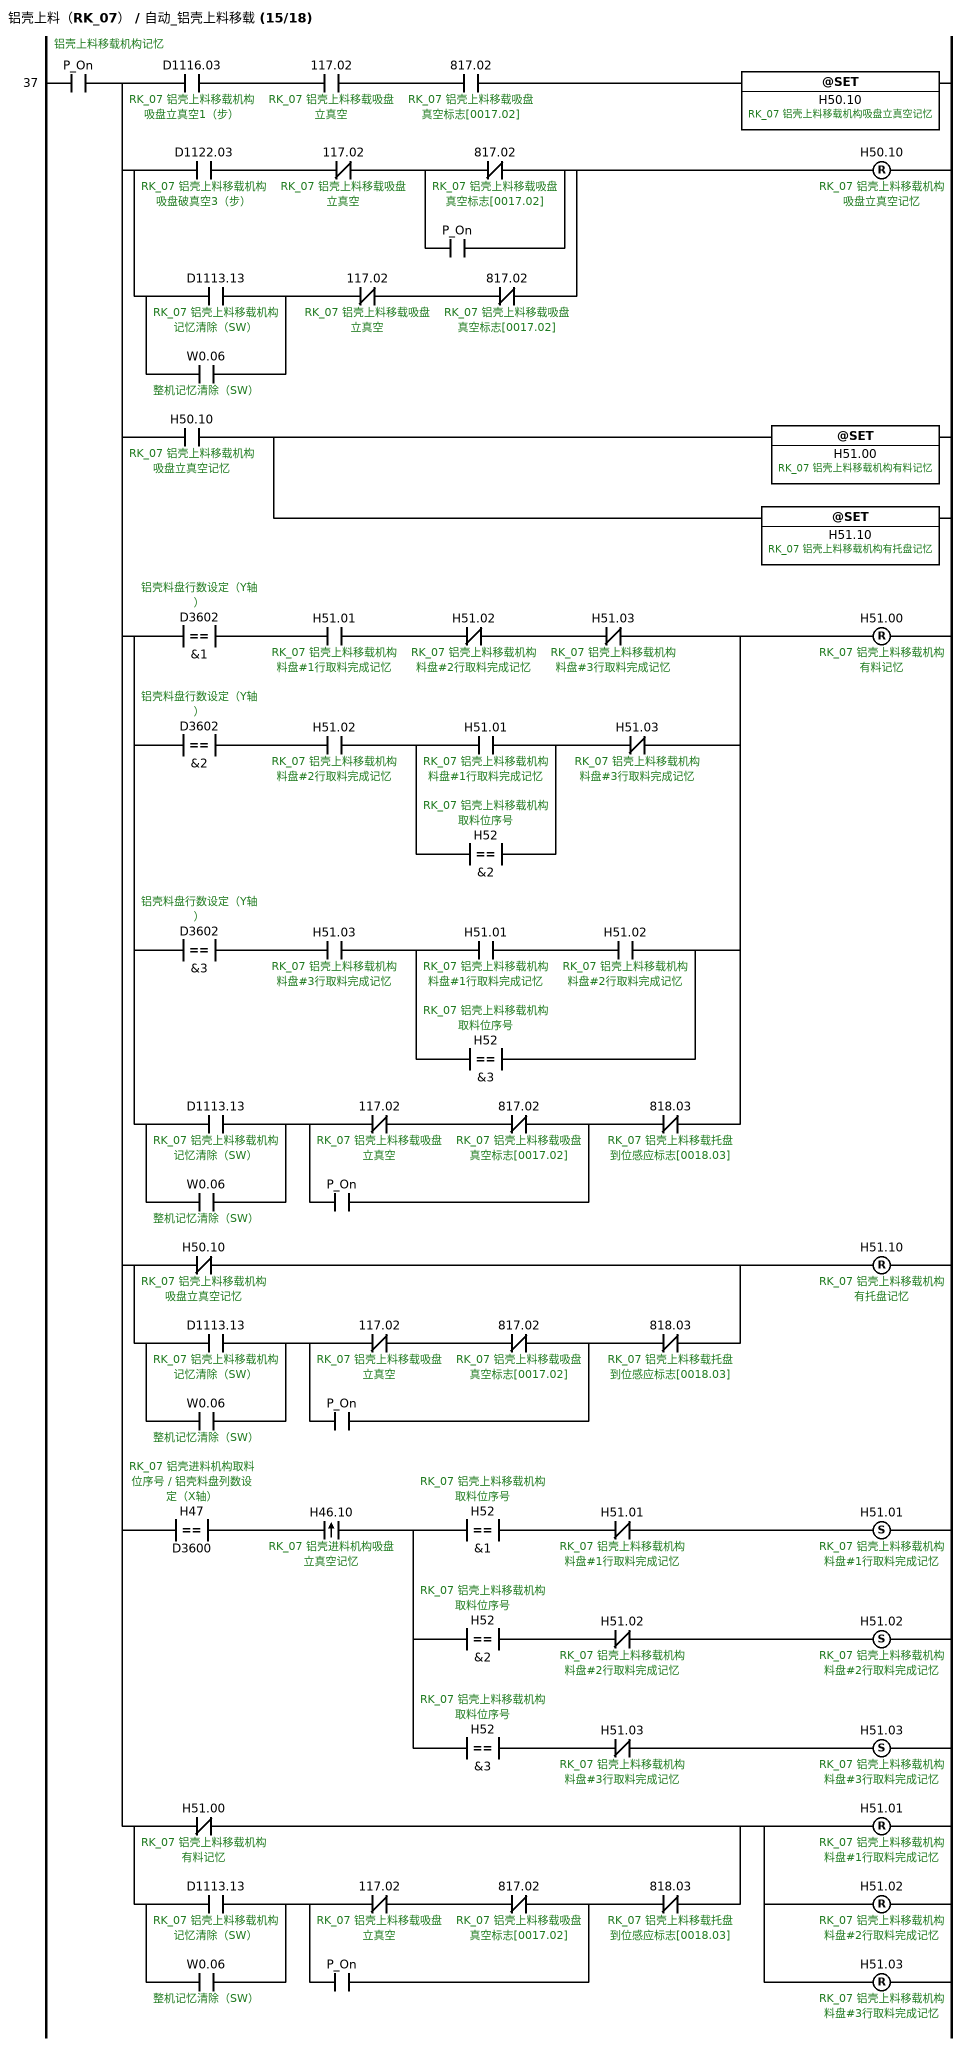
; [picture p600: 铝壳上料（RK_07） / 自动_铝壳上料移载, rungs 37-37]
; rung 37: 铝壳上料移载机构记忆
LD P_On
OUT TR0
AND D1116.03  ; RK_07 铝壳上料移载机构吸盘立真空1（步）
AND 117.02  ; RK_07 铝壳上料移载吸盘立真空
AND 817.02  ; RK_07 铝壳上料移载吸盘真空标志[0017.02]
@SET H50.10  ; RK_07 铝壳上料移载机构吸盘立真空记忆
LD TR0
LD D1122.03  ; RK_07 铝壳上料移载机构吸盘破真空3（步）
ANDNOT 117.02  ; RK_07 铝壳上料移载吸盘立真空
LDNOT 817.02  ; RK_07 铝壳上料移载吸盘真空标志[0017.02]
OR P_On
ANDLD
LD D1113.13  ; RK_07 铝壳上料移载机构记忆清除（SW）
OR W0.06  ; 整机记忆清除（SW）
ANDNOT 117.02  ; RK_07 铝壳上料移载吸盘立真空
ANDNOT 817.02  ; RK_07 铝壳上料移载吸盘真空标志[0017.02]
ORLD
ANDLD
RSET H50.10  ; RK_07 铝壳上料移载机构吸盘立真空记忆
LD TR0
AND H50.10  ; RK_07 铝壳上料移载机构吸盘立真空记忆
@SET H51.00  ; RK_07 铝壳上料移载机构有料记忆
@SET H51.10  ; RK_07 铝壳上料移载机构有托盘记忆
LD TR0
LD=(300) D3602 &1  ; 铝壳料盘行数设定（Y轴）
AND H51.01  ; RK_07 铝壳上料移载机构料盘#1行取料完成记忆
ANDNOT H51.02  ; RK_07 铝壳上料移载机构料盘#2行取料完成记忆
ANDNOT H51.03  ; RK_07 铝壳上料移载机构料盘#3行取料完成记忆
LD=(300) D3602 &2  ; 铝壳料盘行数设定（Y轴）
AND H51.02  ; RK_07 铝壳上料移载机构料盘#2行取料完成记忆
LD H51.01  ; RK_07 铝壳上料移载机构料盘#1行取料完成记忆
OR=(300) H52 &2  ; RK_07 铝壳上料移载机构取料位序号
ANDLD
ANDNOT H51.03  ; RK_07 铝壳上料移载机构料盘#3行取料完成记忆
ORLD
LD=(300) D3602 &3  ; 铝壳料盘行数设定（Y轴）
AND H51.03  ; RK_07 铝壳上料移载机构料盘#3行取料完成记忆
LD H51.01  ; RK_07 铝壳上料移载机构料盘#1行取料完成记忆
AND H51.02  ; RK_07 铝壳上料移载机构料盘#2行取料完成记忆
OR=(300) H52 &3  ; RK_07 铝壳上料移载机构取料位序号
ANDLD
ORLD
LD D1113.13  ; RK_07 铝壳上料移载机构记忆清除（SW）
OR W0.06  ; 整机记忆清除（SW）
LDNOT 117.02  ; RK_07 铝壳上料移载吸盘立真空
ANDNOT 817.02  ; RK_07 铝壳上料移载吸盘真空标志[0017.02]
OR P_On
ANDLD
ANDNOT 818.03  ; RK_07 铝壳上料移载托盘到位感应标志[0018.03]
ORLD
ANDLD
RSET H51.00  ; RK_07 铝壳上料移载机构有料记忆
LD TR0
LDNOT H50.10  ; RK_07 铝壳上料移载机构吸盘立真空记忆
LD D1113.13  ; RK_07 铝壳上料移载机构记忆清除（SW）
OR W0.06  ; 整机记忆清除（SW）
LDNOT 117.02  ; RK_07 铝壳上料移载吸盘立真空
ANDNOT 817.02  ; RK_07 铝壳上料移载吸盘真空标志[0017.02]
OR P_On
ANDLD
ANDNOT 818.03  ; RK_07 铝壳上料移载托盘到位感应标志[0018.03]
ORLD
ANDLD
RSET H51.10  ; RK_07 铝壳上料移载机构有托盘记忆
LD TR0
AND=(300) H47 D3600  ; RK_07 铝壳进料机构取料位序号, 铝壳料盘列数设定（X轴）
@AND H46.10  ; RK_07 铝壳进料机构吸盘立真空记忆
OUT TR1
AND=(300) H52 &1  ; RK_07 铝壳上料移载机构取料位序号
ANDNOT H51.01  ; RK_07 铝壳上料移载机构料盘#1行取料完成记忆
SET H51.01  ; RK_07 铝壳上料移载机构料盘#1行取料完成记忆
LD TR1
AND=(300) H52 &2  ; RK_07 铝壳上料移载机构取料位序号
ANDNOT H51.02  ; RK_07 铝壳上料移载机构料盘#2行取料完成记忆
SET H51.02  ; RK_07 铝壳上料移载机构料盘#2行取料完成记忆
LD TR1
AND=(300) H52 &3  ; RK_07 铝壳上料移载机构取料位序号
ANDNOT H51.03  ; RK_07 铝壳上料移载机构料盘#3行取料完成记忆
SET H51.03  ; RK_07 铝壳上料移载机构料盘#3行取料完成记忆
LD TR0
LDNOT H51.00  ; RK_07 铝壳上料移载机构有料记忆
LD D1113.13  ; RK_07 铝壳上料移载机构记忆清除（SW）
OR W0.06  ; 整机记忆清除（SW）
LDNOT 117.02  ; RK_07 铝壳上料移载吸盘立真空
ANDNOT 817.02  ; RK_07 铝壳上料移载吸盘真空标志[0017.02]
OR P_On
ANDLD
ANDNOT 818.03  ; RK_07 铝壳上料移载托盘到位感应标志[0018.03]
ORLD
ANDLD
RSET H51.01  ; RK_07 铝壳上料移载机构料盘#1行取料完成记忆
RSET H51.02  ; RK_07 铝壳上料移载机构料盘#2行取料完成记忆
RSET H51.03  ; RK_07 铝壳上料移载机构料盘#3行取料完成记忆

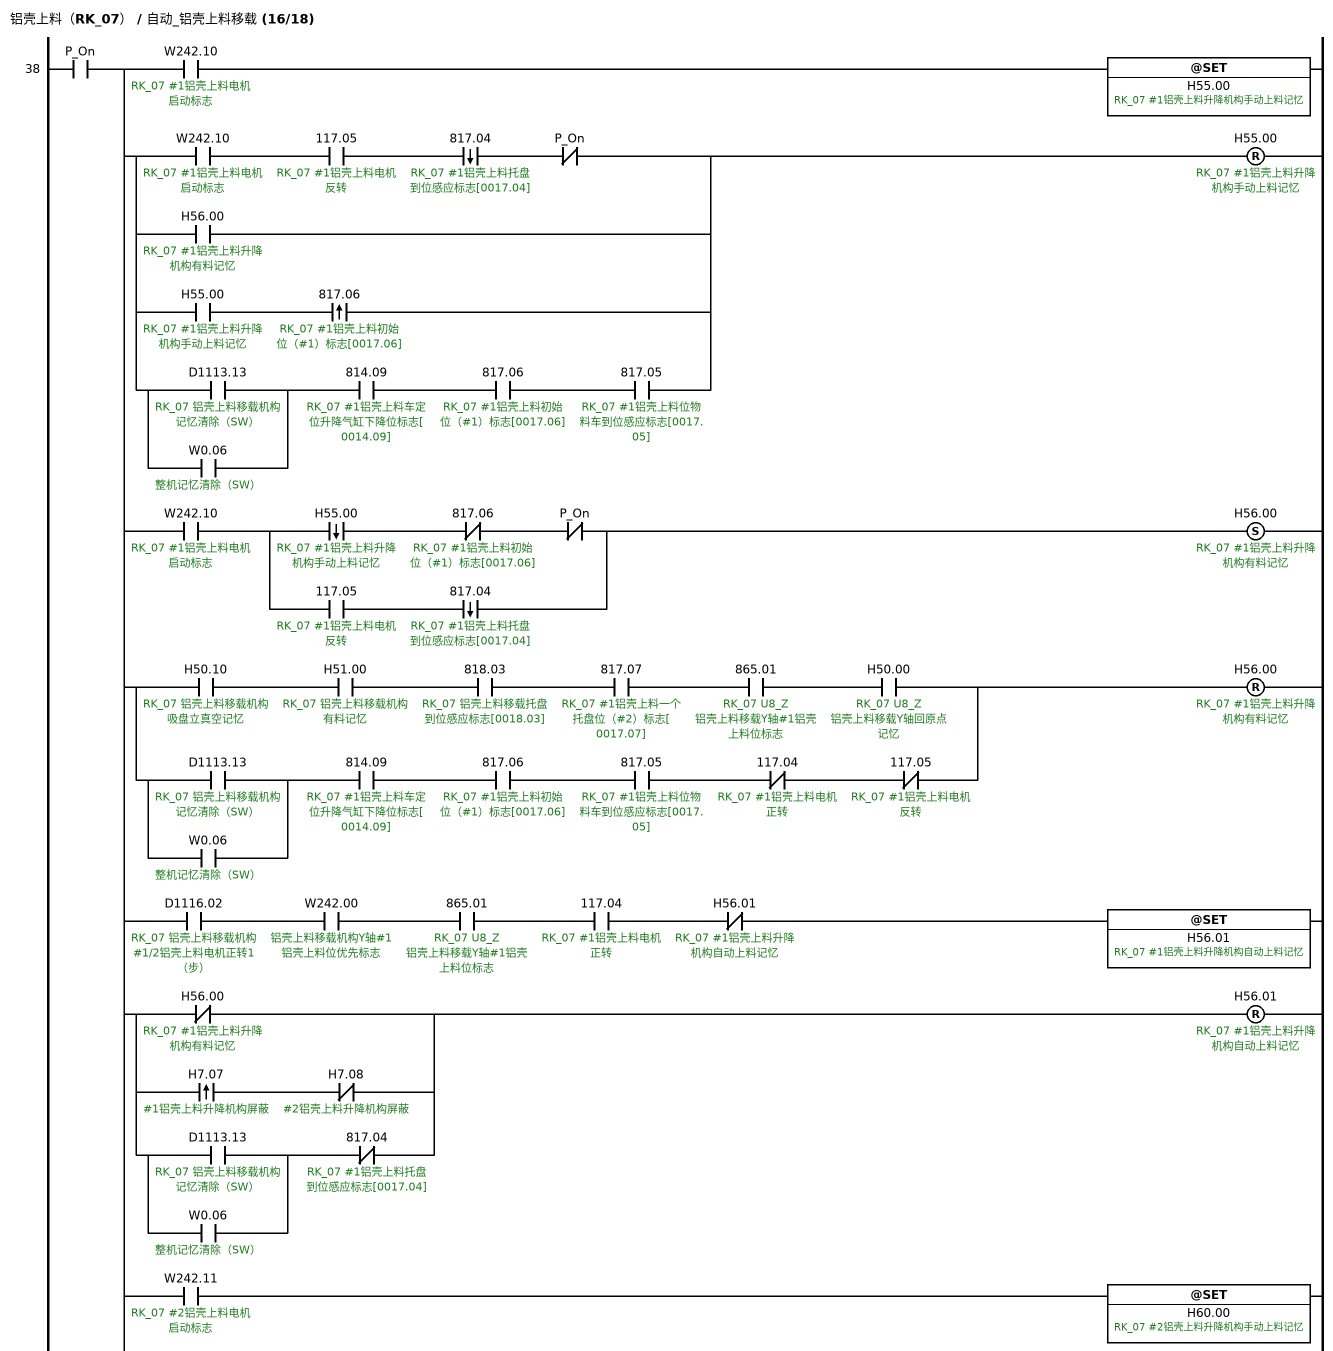

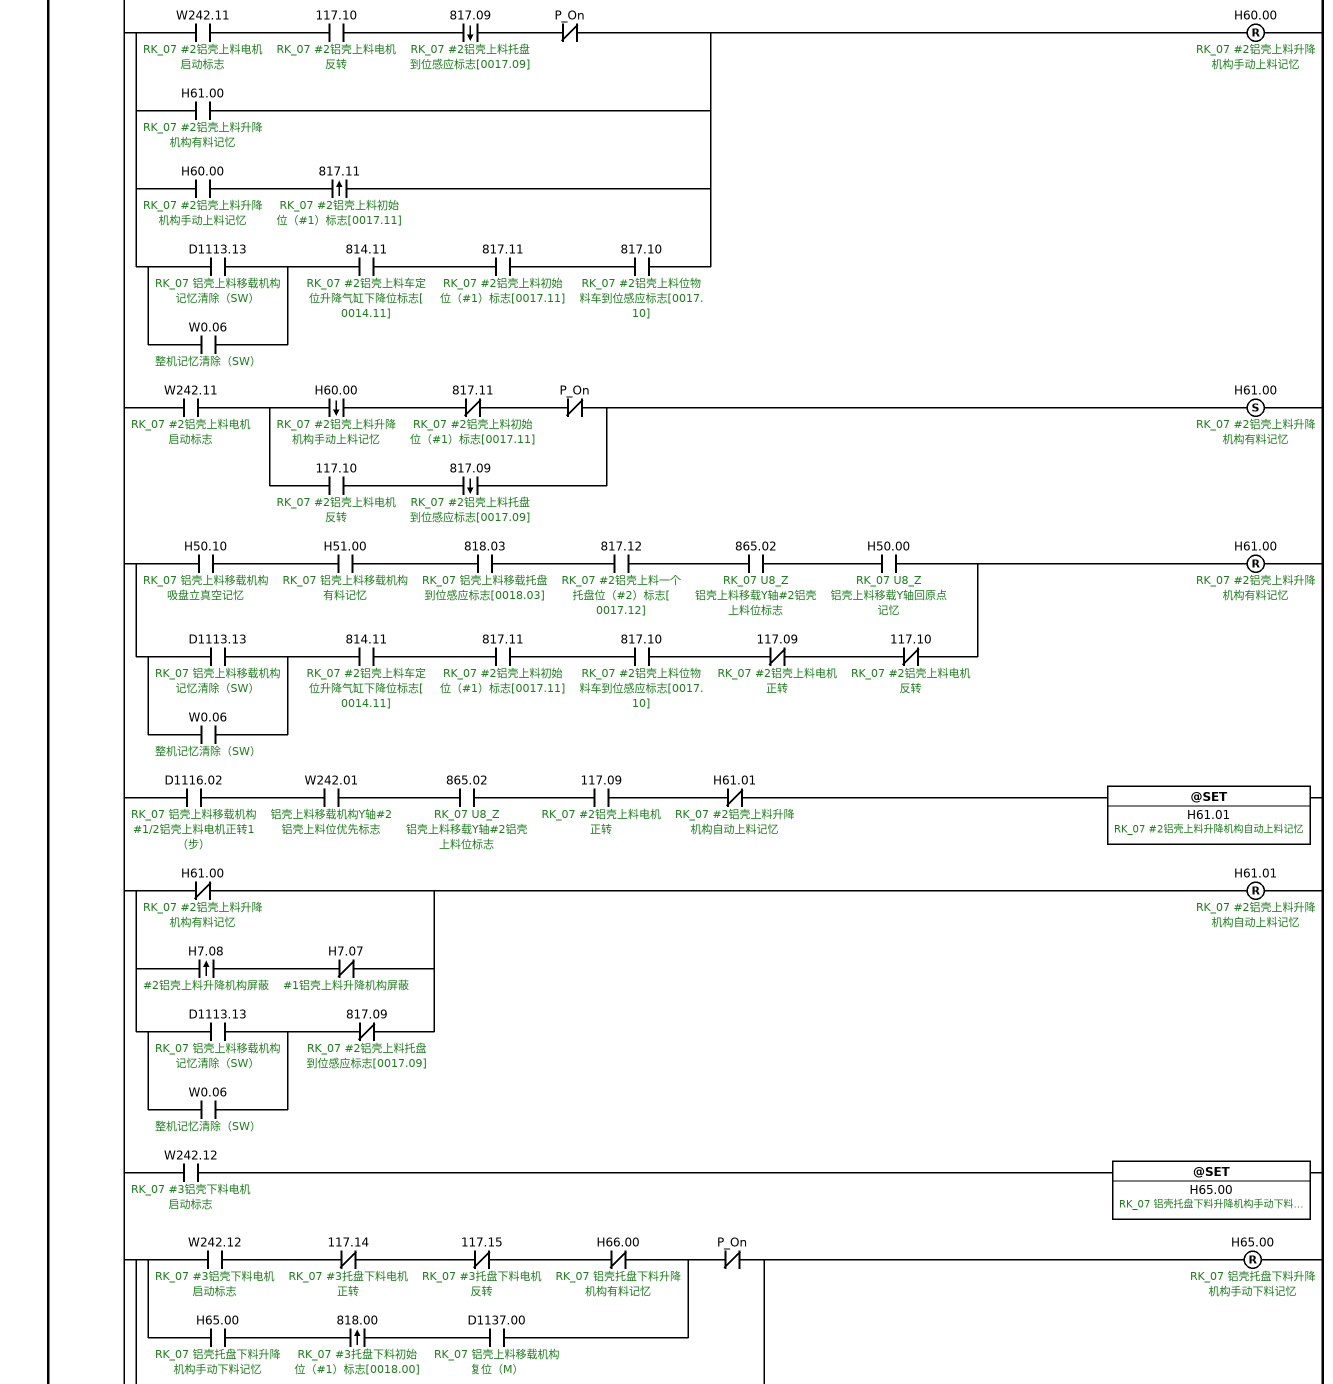

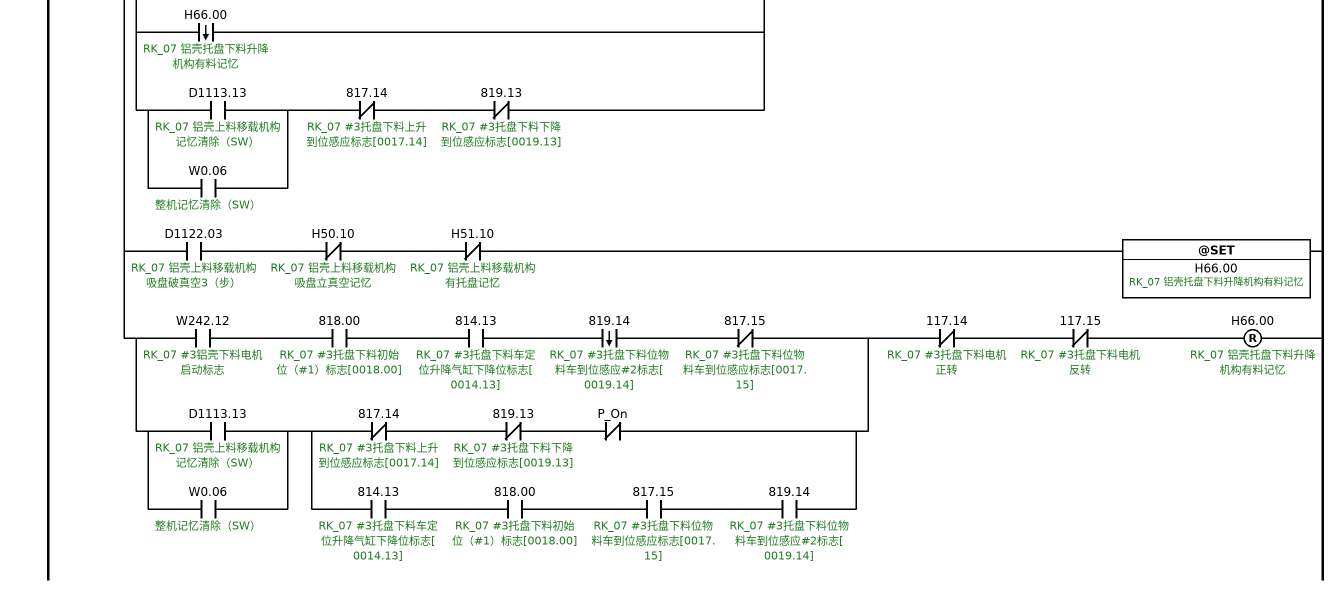
; rung 38
LD P_On
OUT TR0
AND W242.10  ; RK_07 #1铝壳上料电机启动标志
@SET H55.00  ; RK_07 #1铝壳上料升降机构手动上料记忆
LD TR0
LD W242.10  ; RK_07 #1铝壳上料电机启动标志
AND 117.05  ; RK_07 #1铝壳上料电机反转
%AND 817.04  ; RK_07 #1铝壳上料托盘到位感应标志[0017.04]
ANDNOT P_On
OR H56.00  ; RK_07 #1铝壳上料升降机构有料记忆
LD H55.00  ; RK_07 #1铝壳上料升降机构手动上料记忆
@AND 817.06  ; RK_07 #1铝壳上料初始位（#1）标志[0017.06]
ORLD
LD D1113.13  ; RK_07 铝壳上料移载机构记忆清除（SW）
OR W0.06  ; 整机记忆清除（SW）
AND 814.09  ; RK_07 #1铝壳上料车定位升降气缸下降位标志[0014.09]
AND 817.06  ; RK_07 #1铝壳上料初始位（#1）标志[0017.06]
AND 817.05  ; RK_07 #1铝壳上料位物料车到位感应标志[0017.05]
ORLD
ANDLD
RSET H55.00  ; RK_07 #1铝壳上料升降机构手动上料记忆
LD TR0
AND W242.10  ; RK_07 #1铝壳上料电机启动标志
%LD H55.00  ; RK_07 #1铝壳上料升降机构手动上料记忆
ANDNOT 817.06  ; RK_07 #1铝壳上料初始位（#1）标志[0017.06]
ANDNOT P_On
LD 117.05  ; RK_07 #1铝壳上料电机反转
%AND 817.04  ; RK_07 #1铝壳上料托盘到位感应标志[0017.04]
ORLD
ANDLD
SET H56.00  ; RK_07 #1铝壳上料升降机构有料记忆
LD TR0
LD H50.10  ; RK_07 铝壳上料移载机构吸盘立真空记忆
AND H51.00  ; RK_07 铝壳上料移载机构有料记忆
AND 818.03  ; RK_07 铝壳上料移载托盘到位感应标志[0018.03]
AND 817.07  ; RK_07 #1铝壳上料一个托盘位（#2）标志[0017.07]
AND 865.01  ; RK_07 U8_Z 铝壳上料移载Y轴#1铝壳上料位标志
AND H50.00  ; RK_07 U8_Z 铝壳上料移载Y轴回原点记忆
LD D1113.13  ; RK_07 铝壳上料移载机构记忆清除（SW）
OR W0.06  ; 整机记忆清除（SW）
AND 814.09  ; RK_07 #1铝壳上料车定位升降气缸下降位标志[0014.09]
AND 817.06  ; RK_07 #1铝壳上料初始位（#1）标志[0017.06]
AND 817.05  ; RK_07 #1铝壳上料位物料车到位感应标志[0017.05]
ANDNOT 117.04  ; RK_07 #1铝壳上料电机正转
ANDNOT 117.05  ; RK_07 #1铝壳上料电机反转
ORLD
ANDLD
RSET H56.00  ; RK_07 #1铝壳上料升降机构有料记忆
LD TR0
AND D1116.02  ; RK_07 铝壳上料移载机构#1/2铝壳上料电机正转1（步）
AND W242.00  ; 铝壳上料移载机构Y轴#1铝壳上料位优先标志
AND 865.01  ; RK_07 U8_Z 铝壳上料移载Y轴#1铝壳上料位标志
AND 117.04  ; RK_07 #1铝壳上料电机正转
ANDNOT H56.01  ; RK_07 #1铝壳上料升降机构自动上料记忆
@SET H56.01  ; RK_07 #1铝壳上料升降机构自动上料记忆
LD TR0
LDNOT H56.00  ; RK_07 #1铝壳上料升降机构有料记忆
@LD H7.07  ; #1铝壳上料升降机构屏蔽
ANDNOT H7.08  ; #2铝壳上料升降机构屏蔽
ORLD
LD D1113.13  ; RK_07 铝壳上料移载机构记忆清除（SW）
OR W0.06  ; 整机记忆清除（SW）
ANDNOT 817.04  ; RK_07 #1铝壳上料托盘到位感应标志[0017.04]
ORLD
ANDLD
RSET H56.01  ; RK_07 #1铝壳上料升降机构自动上料记忆
LD TR0
AND W242.11  ; RK_07 #2铝壳上料电机启动标志
@SET H60.00  ; RK_07 #2铝壳上料升降机构手动上料记忆
LD TR0
LD W242.11  ; RK_07 #2铝壳上料电机启动标志
AND 117.10  ; RK_07 #2铝壳上料电机反转
%AND 817.09  ; RK_07 #2铝壳上料托盘到位感应标志[0017.09]
ANDNOT P_On
OR H61.00  ; RK_07 #2铝壳上料升降机构有料记忆
LD H60.00  ; RK_07 #2铝壳上料升降机构手动上料记忆
@AND 817.11  ; RK_07 #2铝壳上料初始位（#1）标志[0017.11]
ORLD
LD D1113.13  ; RK_07 铝壳上料移载机构记忆清除（SW）
OR W0.06  ; 整机记忆清除（SW）
AND 814.11  ; RK_07 #2铝壳上料车定位升降气缸下降位标志[0014.11]
AND 817.11  ; RK_07 #2铝壳上料初始位（#1）标志[0017.11]
AND 817.10  ; RK_07 #2铝壳上料位物料车到位感应标志[0017.10]
ORLD
ANDLD
RSET H60.00  ; RK_07 #2铝壳上料升降机构手动上料记忆
LD TR0
AND W242.11  ; RK_07 #2铝壳上料电机启动标志
%LD H60.00  ; RK_07 #2铝壳上料升降机构手动上料记忆
ANDNOT 817.11  ; RK_07 #2铝壳上料初始位（#1）标志[0017.11]
ANDNOT P_On
LD 117.10  ; RK_07 #2铝壳上料电机反转
%AND 817.09  ; RK_07 #2铝壳上料托盘到位感应标志[0017.09]
ORLD
ANDLD
SET H61.00  ; RK_07 #2铝壳上料升降机构有料记忆
LD TR0
LD H50.10  ; RK_07 铝壳上料移载机构吸盘立真空记忆
AND H51.00  ; RK_07 铝壳上料移载机构有料记忆
AND 818.03  ; RK_07 铝壳上料移载托盘到位感应标志[0018.03]
AND 817.12  ; RK_07 #2铝壳上料一个托盘位（#2）标志[0017.12]
AND 865.02  ; RK_07 U8_Z 铝壳上料移载Y轴#2铝壳上料位标志
AND H50.00  ; RK_07 U8_Z 铝壳上料移载Y轴回原点记忆
LD D1113.13  ; RK_07 铝壳上料移载机构记忆清除（SW）
OR W0.06  ; 整机记忆清除（SW）
AND 814.11  ; RK_07 #2铝壳上料车定位升降气缸下降位标志[0014.11]
AND 817.11  ; RK_07 #2铝壳上料初始位（#1）标志[0017.11]
AND 817.10  ; RK_07 #2铝壳上料位物料车到位感应标志[0017.10]
ANDNOT 117.09  ; RK_07 #2铝壳上料电机正转
ANDNOT 117.10  ; RK_07 #2铝壳上料电机反转
ORLD
ANDLD
RSET H61.00  ; RK_07 #2铝壳上料升降机构有料记忆
LD TR0
AND D1116.02  ; RK_07 铝壳上料移载机构#1/2铝壳上料电机正转1（步）
AND W242.01  ; 铝壳上料移载机构Y轴#2铝壳上料位优先标志
AND 865.02  ; RK_07 U8_Z 铝壳上料移载Y轴#2铝壳上料位标志
AND 117.09  ; RK_07 #2铝壳上料电机正转
ANDNOT H61.01  ; RK_07 #2铝壳上料升降机构自动上料记忆
@SET H61.01  ; RK_07 #2铝壳上料升降机构自动上料记忆
LD TR0
LDNOT H61.00  ; RK_07 #2铝壳上料升降机构有料记忆
@LD H7.08  ; #2铝壳上料升降机构屏蔽
ANDNOT H7.07  ; #1铝壳上料升降机构屏蔽
ORLD
LD D1113.13  ; RK_07 铝壳上料移载机构记忆清除（SW）
OR W0.06  ; 整机记忆清除（SW）
ANDNOT 817.09  ; RK_07 #2铝壳上料托盘到位感应标志[0017.09]
ORLD
ANDLD
RSET H61.01  ; RK_07 #2铝壳上料升降机构自动上料记忆
LD TR0
AND W242.12  ; RK_07 #3铝壳下料电机启动标志
@SET H65.00  ; RK_07 铝壳托盘下料升降机构手动下料记忆
LD TR0
LD W242.12  ; RK_07 #3铝壳下料电机启动标志
ANDNOT 117.14  ; RK_07 #3托盘下料电机正转
ANDNOT 117.15  ; RK_07 #3托盘下料电机反转
ANDNOT H66.00  ; RK_07 铝壳托盘下料升降机构有料记忆
LD H65.00  ; RK_07 铝壳托盘下料升降机构手动下料记忆
@AND 818.00  ; RK_07 #3托盘下料初始位（#1）标志[0018.00]
AND D1137.00  ; RK_07 铝壳上料移载机构复位（M）
ORLD
ANDNOT P_On
%OR H66.00  ; RK_07 铝壳托盘下料升降机构有料记忆
LD D1113.13  ; RK_07 铝壳上料移载机构记忆清除（SW）
OR W0.06  ; 整机记忆清除（SW）
ANDNOT 817.14  ; RK_07 #3托盘下料上升到位感应标志[0017.14]
ANDNOT 819.13  ; RK_07 #3托盘下料下降到位感应标志[0019.13]
ORLD
ANDLD
RSET H65.00  ; RK_07 铝壳托盘下料升降机构手动下料记忆
LD TR0
AND D1122.03  ; RK_07 铝壳上料移载机构吸盘破真空3（步）
ANDNOT H50.10  ; RK_07 铝壳上料移载机构吸盘立真空记忆
ANDNOT H51.10  ; RK_07 铝壳上料移载机构有托盘记忆
@SET H66.00  ; RK_07 铝壳托盘下料升降机构有料记忆
LD TR0
LD W242.12  ; RK_07 #3铝壳下料电机启动标志
AND 818.00  ; RK_07 #3托盘下料初始位（#1）标志[0018.00]
AND 814.13  ; RK_07 #3托盘下料车定位升降气缸下降位标志[0014.13]
%AND 819.14  ; RK_07 #3托盘下料位物料车到位感应#2标志[0019.14]
ANDNOT 817.15  ; RK_07 #3托盘下料位物料车到位感应标志[0017.15]
LD D1113.13  ; RK_07 铝壳上料移载机构记忆清除（SW）
OR W0.06  ; 整机记忆清除（SW）
LDNOT 817.14  ; RK_07 #3托盘下料上升到位感应标志[0017.14]
ANDNOT 819.13  ; RK_07 #3托盘下料下降到位感应标志[0019.13]
ANDNOT P_On
LD 814.13  ; RK_07 #3托盘下料车定位升降气缸下降位标志[0014.13]
AND 818.00  ; RK_07 #3托盘下料初始位（#1）标志[0018.00]
AND 817.15  ; RK_07 #3托盘下料位物料车到位感应标志[0017.15]
AND 819.14  ; RK_07 #3托盘下料位物料车到位感应#2标志[0019.14]
ORLD
ANDLD
ORLD
ANDLD
ANDNOT 117.14  ; RK_07 #3托盘下料电机正转
ANDNOT 117.15  ; RK_07 #3托盘下料电机反转
RSET H66.00  ; RK_07 铝壳托盘下料升降机构有料记忆

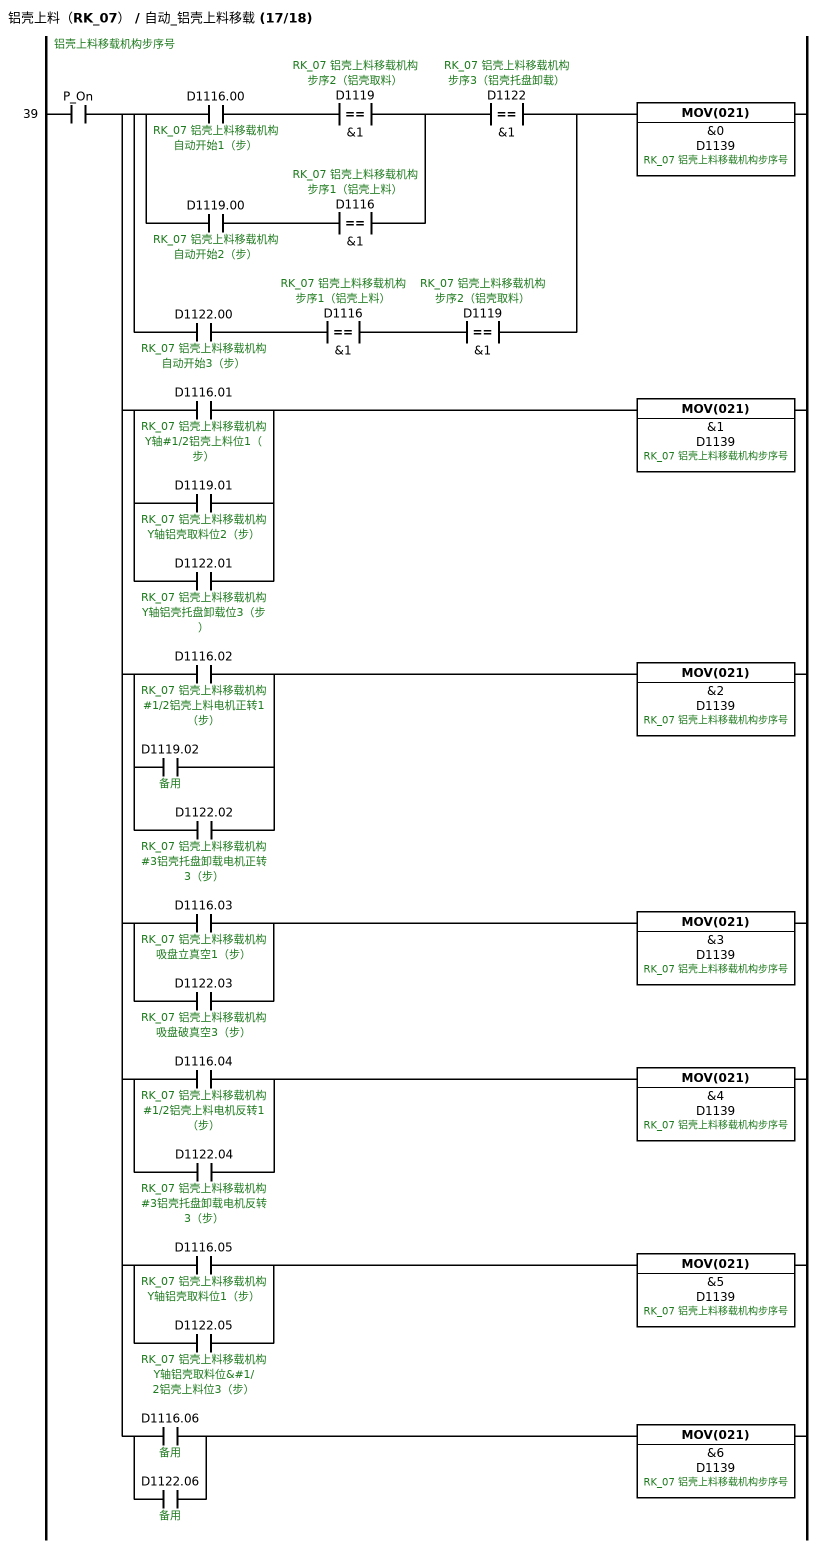
; rung 39: 铝壳上料移载机构步序号
LD P_On
OUT TR0
LD D1116.00  ; RK_07 铝壳上料移载机构自动开始1（步）
AND=(300) D1119 &1  ; RK_07 铝壳上料移载机构步序2（铝壳取料）
LD D1119.00  ; RK_07 铝壳上料移载机构自动开始2（步）
AND=(300) D1116 &1  ; RK_07 铝壳上料移载机构步序1（铝壳上料）
ORLD
AND=(300) D1122 &1  ; RK_07 铝壳上料移载机构步序3（铝壳托盘卸载）
LD D1122.00  ; RK_07 铝壳上料移载机构自动开始3（步）
AND=(300) D1116 &1  ; RK_07 铝壳上料移载机构步序1（铝壳上料）
AND=(300) D1119 &1  ; RK_07 铝壳上料移载机构步序2（铝壳取料）
ORLD
ANDLD
MOV(021) &0 D1139  ; RK_07 铝壳上料移载机构步序号
LD TR0
LD D1116.01  ; RK_07 铝壳上料移载机构Y轴#1/2铝壳上料位1（步）
OR D1119.01  ; RK_07 铝壳上料移载机构Y轴铝壳取料位2（步）
OR D1122.01  ; RK_07 铝壳上料移载机构Y轴铝壳托盘卸载位3（步）
ANDLD
MOV(021) &1 D1139  ; RK_07 铝壳上料移载机构步序号
LD TR0
LD D1116.02  ; RK_07 铝壳上料移载机构#1/2铝壳上料电机正转1（步）
OR D1119.02  ; 备用
OR D1122.02  ; RK_07 铝壳上料移载机构#3铝壳托盘卸载电机正转3（步）
ANDLD
MOV(021) &2 D1139  ; RK_07 铝壳上料移载机构步序号
LD TR0
LD D1116.03  ; RK_07 铝壳上料移载机构吸盘立真空1（步）
OR D1122.03  ; RK_07 铝壳上料移载机构吸盘破真空3（步）
ANDLD
MOV(021) &3 D1139  ; RK_07 铝壳上料移载机构步序号
LD TR0
LD D1116.04  ; RK_07 铝壳上料移载机构#1/2铝壳上料电机反转1（步）
OR D1122.04  ; RK_07 铝壳上料移载机构#3铝壳托盘卸载电机反转3（步）
ANDLD
MOV(021) &4 D1139  ; RK_07 铝壳上料移载机构步序号
LD TR0
LD D1116.05  ; RK_07 铝壳上料移载机构Y轴铝壳取料位1（步）
OR D1122.05  ; RK_07 铝壳上料移载机构Y轴铝壳取料位&#1/2铝壳上料位3（步）
ANDLD
MOV(021) &5 D1139  ; RK_07 铝壳上料移载机构步序号
LD TR0
LD D1116.06  ; 备用
OR D1122.06  ; 备用
ANDLD
MOV(021) &6 D1139  ; RK_07 铝壳上料移载机构步序号

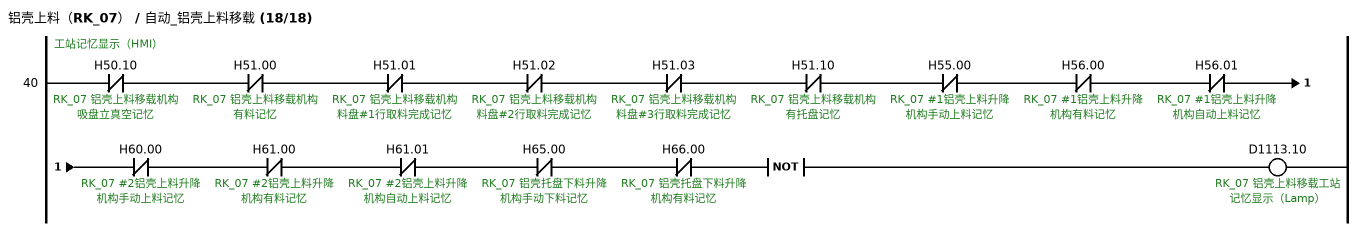
; rung 40: 工站记忆显示（HMI）
LDNOT H50.10  ; RK_07 铝壳上料移载机构吸盘立真空记忆
ANDNOT H51.00  ; RK_07 铝壳上料移载机构有料记忆
ANDNOT H51.01  ; RK_07 铝壳上料移载机构料盘#1行取料完成记忆
ANDNOT H51.02  ; RK_07 铝壳上料移载机构料盘#2行取料完成记忆
ANDNOT H51.03  ; RK_07 铝壳上料移载机构料盘#3行取料完成记忆
ANDNOT H51.10  ; RK_07 铝壳上料移载机构有托盘记忆
ANDNOT H55.00  ; RK_07 #1铝壳上料升降机构手动上料记忆
ANDNOT H56.00  ; RK_07 #1铝壳上料升降机构有料记忆
ANDNOT H56.01  ; RK_07 #1铝壳上料升降机构自动上料记忆
ANDNOT H60.00  ; RK_07 #2铝壳上料升降机构手动上料记忆
ANDNOT H61.00  ; RK_07 #2铝壳上料升降机构有料记忆
ANDNOT H61.01  ; RK_07 #2铝壳上料升降机构自动上料记忆
ANDNOT H65.00  ; RK_07 铝壳托盘下料升降机构手动下料记忆
ANDNOT H66.00  ; RK_07 铝壳托盘下料升降机构有料记忆
NOT(520)
OUT D1113.10  ; RK_07 铝壳上料移载工站记忆显示（Lamp）

### Section 自动_铝壳上下料升降

### Section 复位

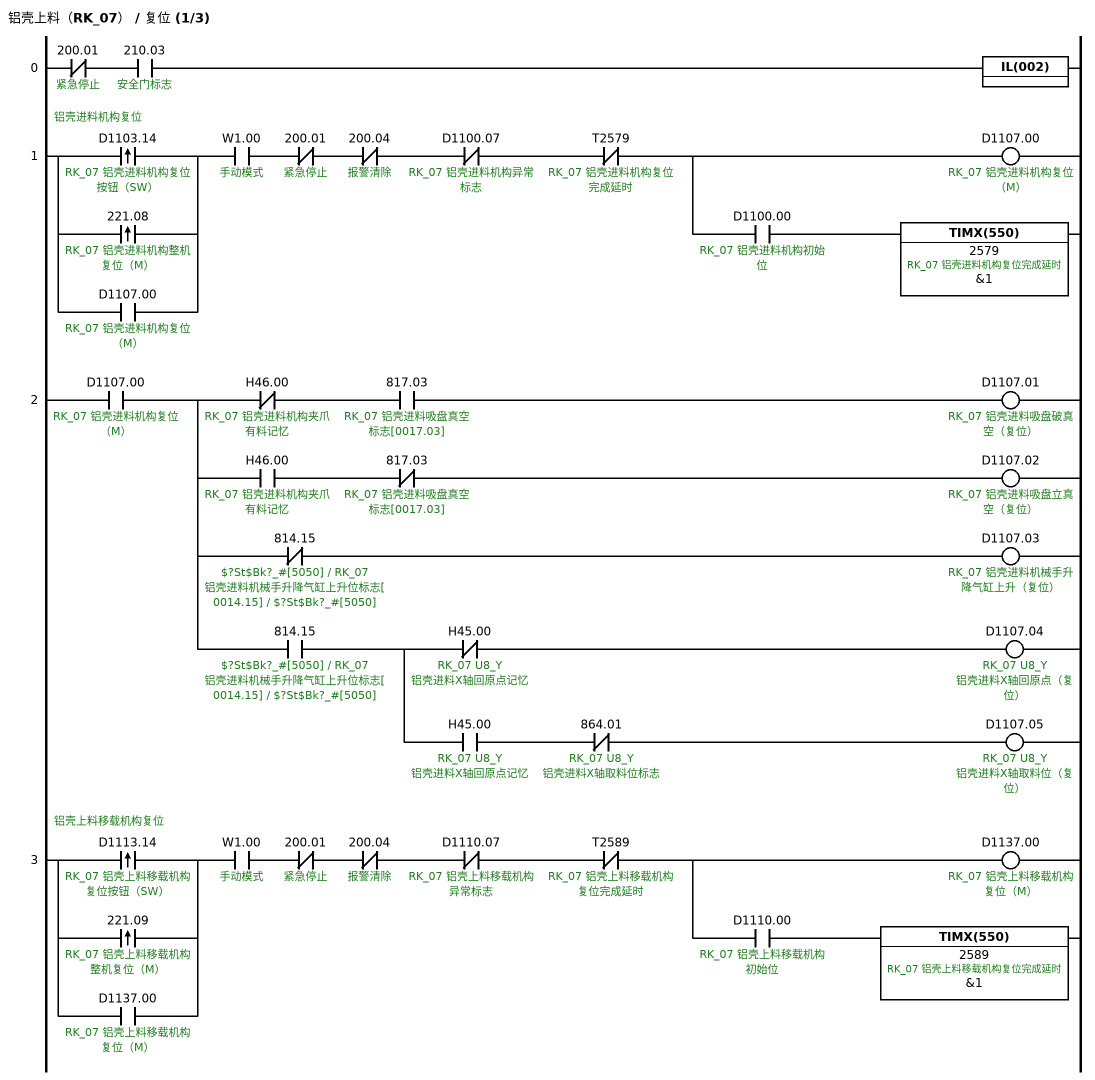
; rung 0
LDNOT 200.01  ; 紧急停止
AND 210.03  ; 安全门标志
IL(002)
; rung 1: 铝壳进料机构复位
@LD D1103.14  ; RK_07 铝壳进料机构复位按钮（SW）
@OR 221.08  ; RK_07 铝壳进料机构整机复位（M）
OR D1107.00  ; RK_07 铝壳进料机构复位（M）
AND W1.00  ; 手动模式
ANDNOT 200.01  ; 紧急停止
ANDNOT 200.04  ; 报警清除
ANDNOT D1100.07  ; RK_07 铝壳进料机构异常标志
ANDNOT T2579  ; RK_07 铝壳进料机构复位完成延时
OUT D1107.00  ; RK_07 铝壳进料机构复位（M）
AND D1100.00  ; RK_07 铝壳进料机构初始位
TIMX(550) 2579 &1  ; RK_07 铝壳进料机构复位完成延时
; rung 2
LD D1107.00  ; RK_07 铝壳进料机构复位（M）
OUT TR0
ANDNOT H46.00  ; RK_07 铝壳进料机构夹爪有料记忆
AND 817.03  ; RK_07 铝壳进料吸盘真空标志[0017.03]
OUT D1107.01  ; RK_07 铝壳进料吸盘破真空（复位）
LD TR0
AND H46.00  ; RK_07 铝壳进料机构夹爪有料记忆
ANDNOT 817.03  ; RK_07 铝壳进料吸盘真空标志[0017.03]
OUT D1107.02  ; RK_07 铝壳进料吸盘立真空（复位）
LD TR0
ANDNOT 814.15  ; $?St$Bk?_#[5050] / RK_07 铝壳进料机械手升降气缸上升位标志[0014.15] / $?St$Bk?_#[5050]
OUT D1107.03  ; RK_07 铝壳进料机械手升降气缸上升（复位）
LD TR0
AND 814.15  ; $?St$Bk?_#[5050] / RK_07 铝壳进料机械手升降气缸上升位标志[0014.15] / $?St$Bk?_#[5050]
OUT TR0
ANDNOT H45.00  ; RK_07 U8_Y 铝壳进料X轴回原点记忆
OUT D1107.04  ; RK_07 U8_Y 铝壳进料X轴回原点（复位）
LD TR0
AND H45.00  ; RK_07 U8_Y 铝壳进料X轴回原点记忆
ANDNOT 864.01  ; RK_07 U8_Y 铝壳进料X轴取料位标志
OUT D1107.05  ; RK_07 U8_Y 铝壳进料X轴取料位（复位）
; rung 3: 铝壳上料移载机构复位
@LD D1113.14  ; RK_07 铝壳上料移载机构复位按钮（SW）
@OR 221.09  ; RK_07 铝壳上料移载机构整机复位（M）
OR D1137.00  ; RK_07 铝壳上料移载机构复位（M）
AND W1.00  ; 手动模式
ANDNOT 200.01  ; 紧急停止
ANDNOT 200.04  ; 报警清除
ANDNOT D1110.07  ; RK_07 铝壳上料移载机构异常标志
ANDNOT T2589  ; RK_07 铝壳上料移载机构复位完成延时
OUT D1137.00  ; RK_07 铝壳上料移载机构复位（M）
AND D1110.00  ; RK_07 铝壳上料移载机构初始位
TIMX(550) 2589 &1  ; RK_07 铝壳上料移载机构复位完成延时

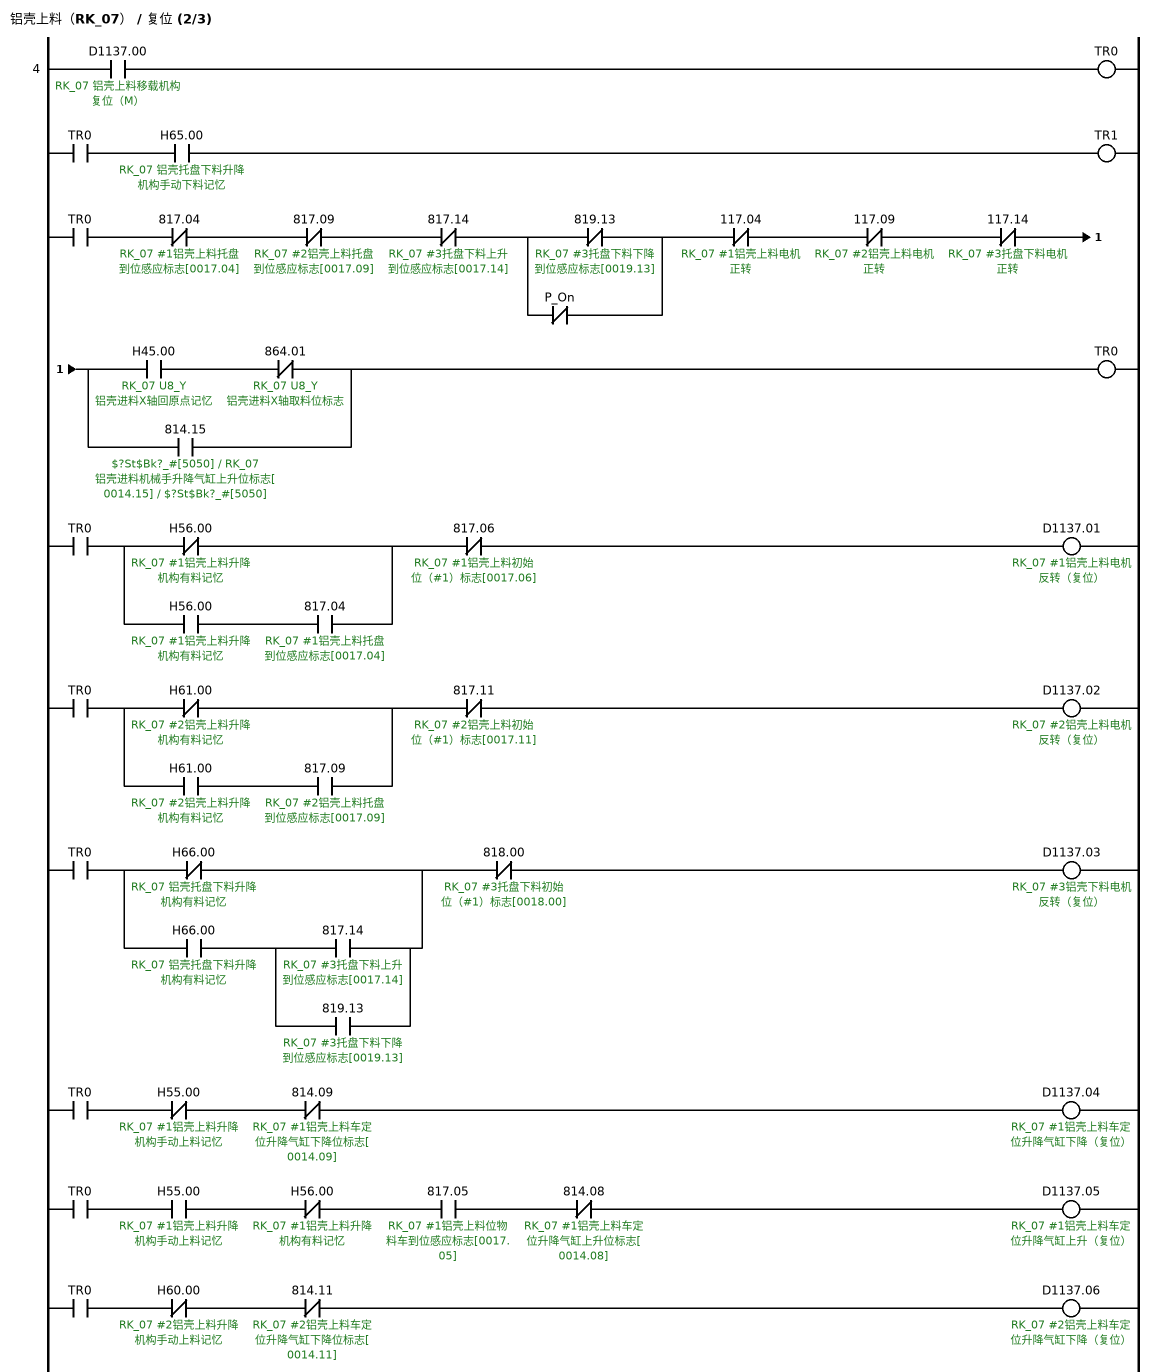

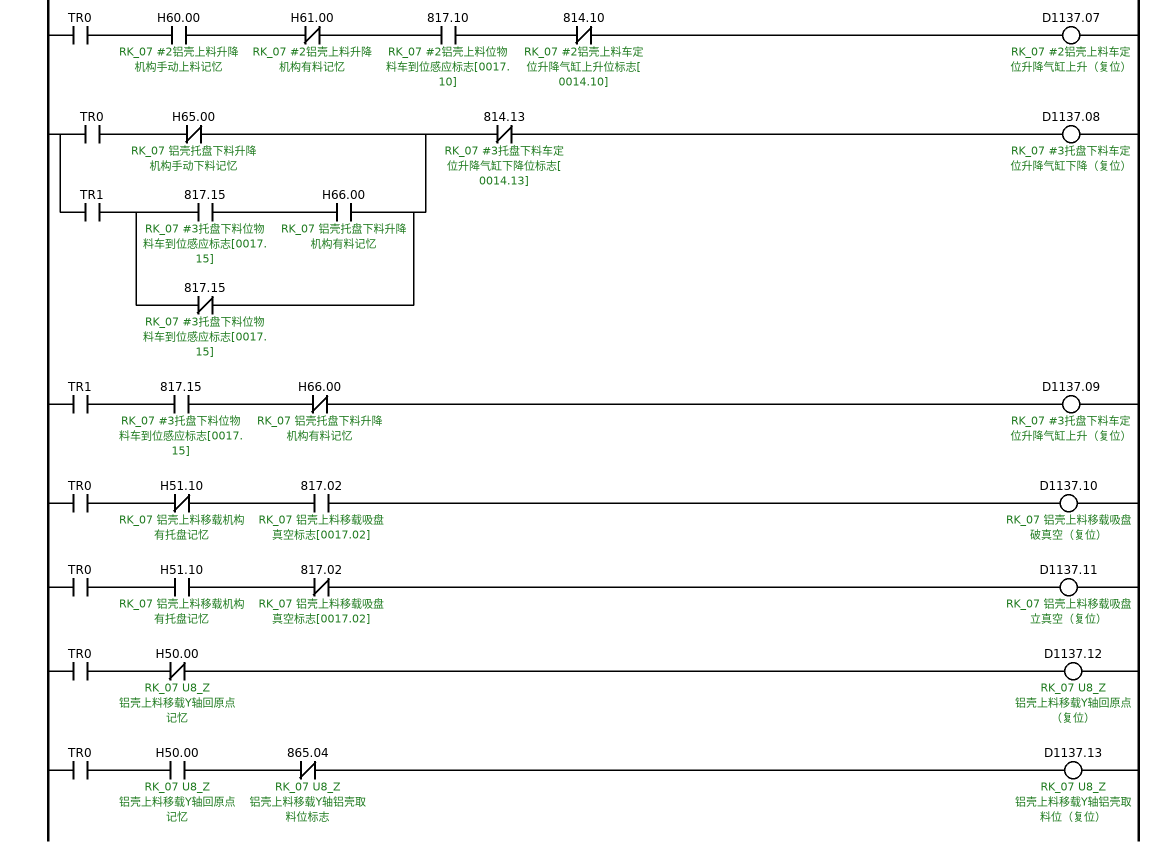
; rung 4
LD D1137.00  ; RK_07 铝壳上料移载机构复位（M）
OUT TR0
LDNOT H56.00  ; RK_07 #1铝壳上料升降机构有料记忆
LD H56.00  ; RK_07 #1铝壳上料升降机构有料记忆
AND 817.04  ; RK_07 #1铝壳上料托盘到位感应标志[0017.04]
ORLD
ANDLD
ANDNOT 817.06  ; RK_07 #1铝壳上料初始位（#1）标志[0017.06]
OUT D1137.01  ; RK_07 #1铝壳上料电机反转（复位）
LD TR0
LDNOT H61.00  ; RK_07 #2铝壳上料升降机构有料记忆
LD H61.00  ; RK_07 #2铝壳上料升降机构有料记忆
AND 817.09  ; RK_07 #2铝壳上料托盘到位感应标志[0017.09]
ORLD
ANDLD
ANDNOT 817.11  ; RK_07 #2铝壳上料初始位（#1）标志[0017.11]
OUT D1137.02  ; RK_07 #2铝壳上料电机反转（复位）
LD TR0
LDNOT H66.00  ; RK_07 铝壳托盘下料升降机构有料记忆
LD H66.00  ; RK_07 铝壳托盘下料升降机构有料记忆
LD 817.14  ; RK_07 #3托盘下料上升到位感应标志[0017.14]
OR 819.13  ; RK_07 #3托盘下料下降到位感应标志[0019.13]
ANDLD
ORLD
ANDLD
ANDNOT 818.00  ; RK_07 #3托盘下料初始位（#1）标志[0018.00]
OUT D1137.03  ; RK_07 #3铝壳下料电机反转（复位）
LD TR0
ANDNOT H55.00  ; RK_07 #1铝壳上料升降机构手动上料记忆
ANDNOT 814.09  ; RK_07 #1铝壳上料车定位升降气缸下降位标志[0014.09]
OUT D1137.04  ; RK_07 #1铝壳上料车定位升降气缸下降（复位）
LD TR0
AND H55.00  ; RK_07 #1铝壳上料升降机构手动上料记忆
ANDNOT H56.00  ; RK_07 #1铝壳上料升降机构有料记忆
AND 817.05  ; RK_07 #1铝壳上料位物料车到位感应标志[0017.05]
ANDNOT 814.08  ; RK_07 #1铝壳上料车定位升降气缸上升位标志[0014.08]
OUT D1137.05  ; RK_07 #1铝壳上料车定位升降气缸上升（复位）
LD TR0
ANDNOT H60.00  ; RK_07 #2铝壳上料升降机构手动上料记忆
ANDNOT 814.11  ; RK_07 #2铝壳上料车定位升降气缸下降位标志[0014.11]
OUT D1137.06  ; RK_07 #2铝壳上料车定位升降气缸下降（复位）
LD TR0
AND H60.00  ; RK_07 #2铝壳上料升降机构手动上料记忆
ANDNOT H61.00  ; RK_07 #2铝壳上料升降机构有料记忆
AND 817.10  ; RK_07 #2铝壳上料位物料车到位感应标志[0017.10]
ANDNOT 814.10  ; RK_07 #2铝壳上料车定位升降气缸上升位标志[0014.10]
OUT D1137.07  ; RK_07 #2铝壳上料车定位升降气缸上升（复位）
LD TR0
ANDNOT H65.00  ; RK_07 铝壳托盘下料升降机构手动下料记忆
LD TR0
AND H65.00  ; RK_07 铝壳托盘下料升降机构手动下料记忆
OUT TR1
LD 817.15  ; RK_07 #3托盘下料位物料车到位感应标志[0017.15]
AND H66.00  ; RK_07 铝壳托盘下料升降机构有料记忆
ORNOT 817.15  ; RK_07 #3托盘下料位物料车到位感应标志[0017.15]
ANDLD
ORLD
ANDNOT 814.13  ; RK_07 #3托盘下料车定位升降气缸下降位标志[0014.13]
OUT D1137.08  ; RK_07 #3托盘下料车定位升降气缸下降（复位）
LD TR1
AND 817.15  ; RK_07 #3托盘下料位物料车到位感应标志[0017.15]
ANDNOT H66.00  ; RK_07 铝壳托盘下料升降机构有料记忆
OUT D1137.09  ; RK_07 #3托盘下料车定位升降气缸上升（复位）
LD TR0
ANDNOT H51.10  ; RK_07 铝壳上料移载机构有托盘记忆
AND 817.02  ; RK_07 铝壳上料移载吸盘真空标志[0017.02]
OUT D1137.10  ; RK_07 铝壳上料移载吸盘破真空（复位）
LD TR0
AND H51.10  ; RK_07 铝壳上料移载机构有托盘记忆
ANDNOT 817.02  ; RK_07 铝壳上料移载吸盘真空标志[0017.02]
OUT D1137.11  ; RK_07 铝壳上料移载吸盘立真空（复位）
LD TR0
ANDNOT 817.04  ; RK_07 #1铝壳上料托盘到位感应标志[0017.04]
ANDNOT 817.09  ; RK_07 #2铝壳上料托盘到位感应标志[0017.09]
ANDNOT 817.14  ; RK_07 #3托盘下料上升到位感应标志[0017.14]
LDNOT 819.13  ; RK_07 #3托盘下料下降到位感应标志[0019.13]
ORNOT P_On
ANDLD
ANDNOT 117.04  ; RK_07 #1铝壳上料电机正转
ANDNOT 117.09  ; RK_07 #2铝壳上料电机正转
ANDNOT 117.14  ; RK_07 #3托盘下料电机正转
LD H45.00  ; RK_07 U8_Y 铝壳进料X轴回原点记忆
ANDNOT 864.01  ; RK_07 U8_Y 铝壳进料X轴取料位标志
OR 814.15  ; $?St$Bk?_#[5050] / RK_07 铝壳进料机械手升降气缸上升位标志[0014.15] / $?St$Bk?_#[5050]
ANDLD
OUT TR0
ANDNOT H50.00  ; RK_07 U8_Z 铝壳上料移载Y轴回原点记忆
OUT D1137.12  ; RK_07 U8_Z 铝壳上料移载Y轴回原点（复位）
LD TR0
AND H50.00  ; RK_07 U8_Z 铝壳上料移载Y轴回原点记忆
ANDNOT 865.04  ; RK_07 U8_Z 铝壳上料移载Y轴铝壳取料位标志
OUT D1137.13  ; RK_07 U8_Z 铝壳上料移载Y轴铝壳取料位（复位）

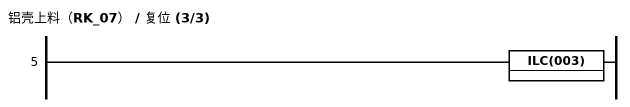
; rung 5
ILC(003)

### Section 指示灯

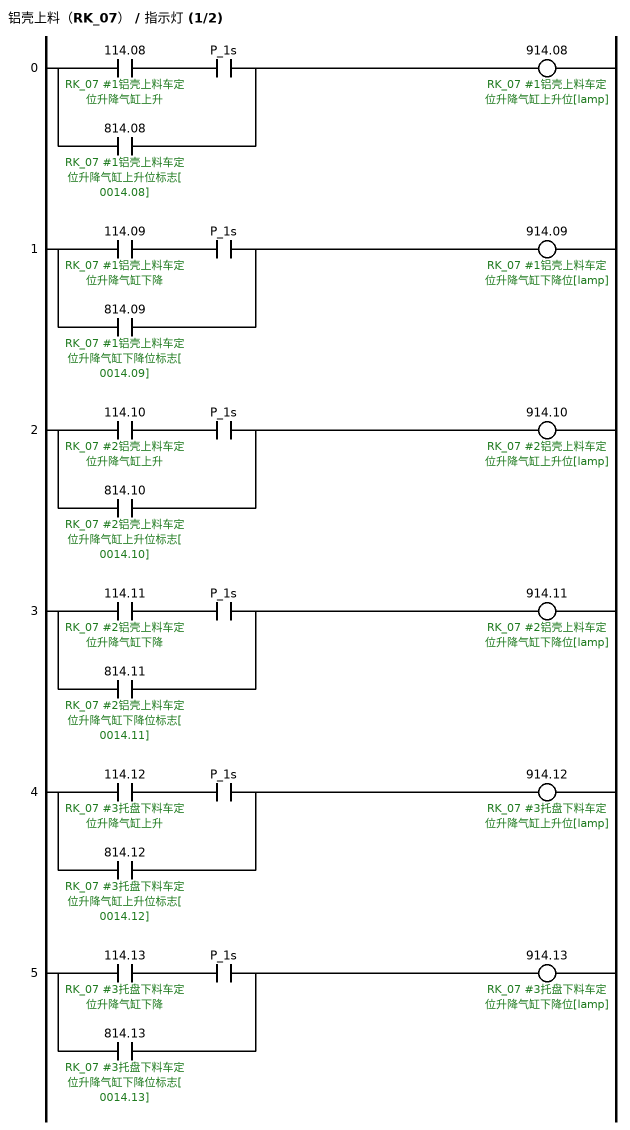
; rung 0
LD 114.08  ; RK_07 #1铝壳上料车定位升降气缸上升
AND P_1s
OR 814.08  ; RK_07 #1铝壳上料车定位升降气缸上升位标志[0014.08]
OUT 914.08  ; RK_07 #1铝壳上料车定位升降气缸上升位[lamp]
; rung 1
LD 114.09  ; RK_07 #1铝壳上料车定位升降气缸下降
AND P_1s
OR 814.09  ; RK_07 #1铝壳上料车定位升降气缸下降位标志[0014.09]
OUT 914.09  ; RK_07 #1铝壳上料车定位升降气缸下降位[lamp]
; rung 2
LD 114.10  ; RK_07 #2铝壳上料车定位升降气缸上升
AND P_1s
OR 814.10  ; RK_07 #2铝壳上料车定位升降气缸上升位标志[0014.10]
OUT 914.10  ; RK_07 #2铝壳上料车定位升降气缸上升位[lamp]
; rung 3
LD 114.11  ; RK_07 #2铝壳上料车定位升降气缸下降
AND P_1s
OR 814.11  ; RK_07 #2铝壳上料车定位升降气缸下降位标志[0014.11]
OUT 914.11  ; RK_07 #2铝壳上料车定位升降气缸下降位[lamp]
; rung 4
LD 114.12  ; RK_07 #3托盘下料车定位升降气缸上升
AND P_1s
OR 814.12  ; RK_07 #3托盘下料车定位升降气缸上升位标志[0014.12]
OUT 914.12  ; RK_07 #3托盘下料车定位升降气缸上升位[lamp]
; rung 5
LD 114.13  ; RK_07 #3托盘下料车定位升降气缸下降
AND P_1s
OR 814.13  ; RK_07 #3托盘下料车定位升降气缸下降位标志[0014.13]
OUT 914.13  ; RK_07 #3托盘下料车定位升降气缸下降位[lamp]

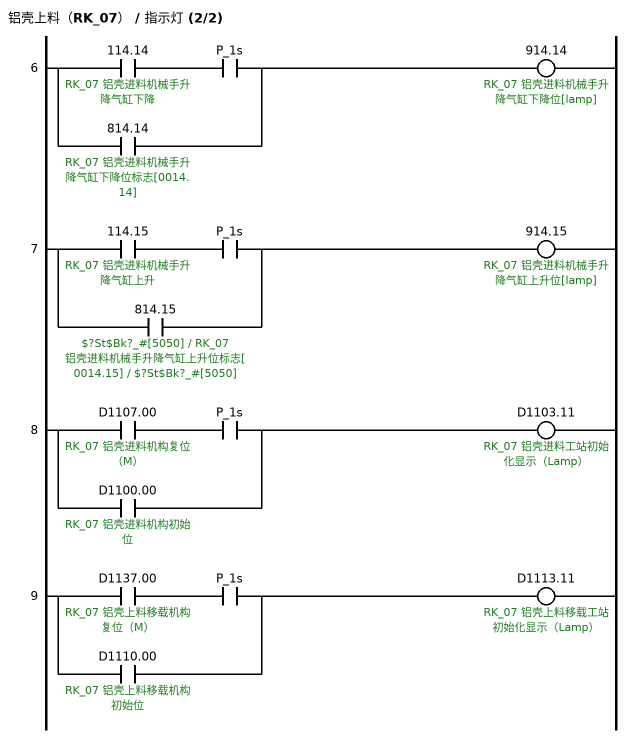
; rung 6
LD 114.14  ; RK_07 铝壳进料机械手升降气缸下降
AND P_1s
OR 814.14  ; RK_07 铝壳进料机械手升降气缸下降位标志[0014.14]
OUT 914.14  ; RK_07 铝壳进料机械手升降气缸下降位[lamp]
; rung 7
LD 114.15  ; RK_07 铝壳进料机械手升降气缸上升
AND P_1s
OR 814.15  ; $?St$Bk?_#[5050] / RK_07 铝壳进料机械手升降气缸上升位标志[0014.15] / $?St$Bk?_#[5050]
OUT 914.15  ; RK_07 铝壳进料机械手升降气缸上升位[lamp]
; rung 8
LD D1107.00  ; RK_07 铝壳进料机构复位（M）
AND P_1s
OR D1100.00  ; RK_07 铝壳进料机构初始位
OUT D1103.11  ; RK_07 铝壳进料工站初始化显示（Lamp）
; rung 9
LD D1137.00  ; RK_07 铝壳上料移载机构复位（M）
AND P_1s
OR D1110.00  ; RK_07 铝壳上料移载机构初始位
OUT D1113.11  ; RK_07 铝壳上料移载工站初始化显示（Lamp）

### Section 外部输出

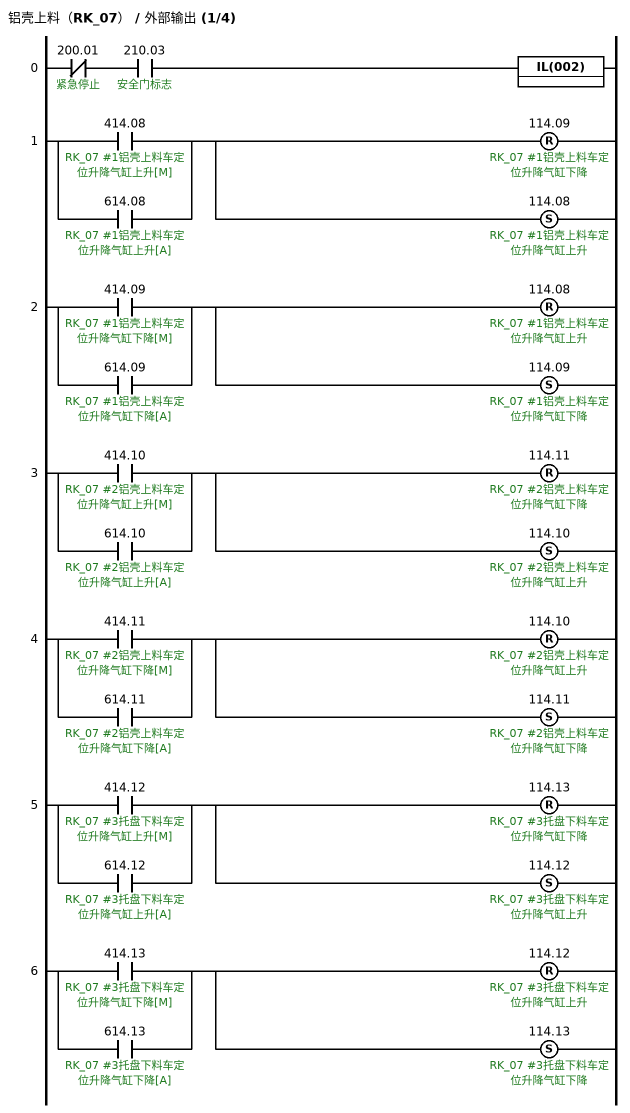
; rung 0
LDNOT 200.01  ; 紧急停止
AND 210.03  ; 安全门标志
IL(002)
; rung 1
LD 414.08  ; RK_07 #1铝壳上料车定位升降气缸上升[M]
OR 614.08  ; RK_07 #1铝壳上料车定位升降气缸上升[A]
RSET 114.09  ; RK_07 #1铝壳上料车定位升降气缸下降
SET 114.08  ; RK_07 #1铝壳上料车定位升降气缸上升
; rung 2
LD 414.09  ; RK_07 #1铝壳上料车定位升降气缸下降[M]
OR 614.09  ; RK_07 #1铝壳上料车定位升降气缸下降[A]
RSET 114.08  ; RK_07 #1铝壳上料车定位升降气缸上升
SET 114.09  ; RK_07 #1铝壳上料车定位升降气缸下降
; rung 3
LD 414.10  ; RK_07 #2铝壳上料车定位升降气缸上升[M]
OR 614.10  ; RK_07 #2铝壳上料车定位升降气缸上升[A]
RSET 114.11  ; RK_07 #2铝壳上料车定位升降气缸下降
SET 114.10  ; RK_07 #2铝壳上料车定位升降气缸上升
; rung 4
LD 414.11  ; RK_07 #2铝壳上料车定位升降气缸下降[M]
OR 614.11  ; RK_07 #2铝壳上料车定位升降气缸下降[A]
RSET 114.10  ; RK_07 #2铝壳上料车定位升降气缸上升
SET 114.11  ; RK_07 #2铝壳上料车定位升降气缸下降
; rung 5
LD 414.12  ; RK_07 #3托盘下料车定位升降气缸上升[M]
OR 614.12  ; RK_07 #3托盘下料车定位升降气缸上升[A]
RSET 114.13  ; RK_07 #3托盘下料车定位升降气缸下降
SET 114.12  ; RK_07 #3托盘下料车定位升降气缸上升
; rung 6
LD 414.13  ; RK_07 #3托盘下料车定位升降气缸下降[M]
OR 614.13  ; RK_07 #3托盘下料车定位升降气缸下降[A]
RSET 114.12  ; RK_07 #3托盘下料车定位升降气缸上升
SET 114.13  ; RK_07 #3托盘下料车定位升降气缸下降

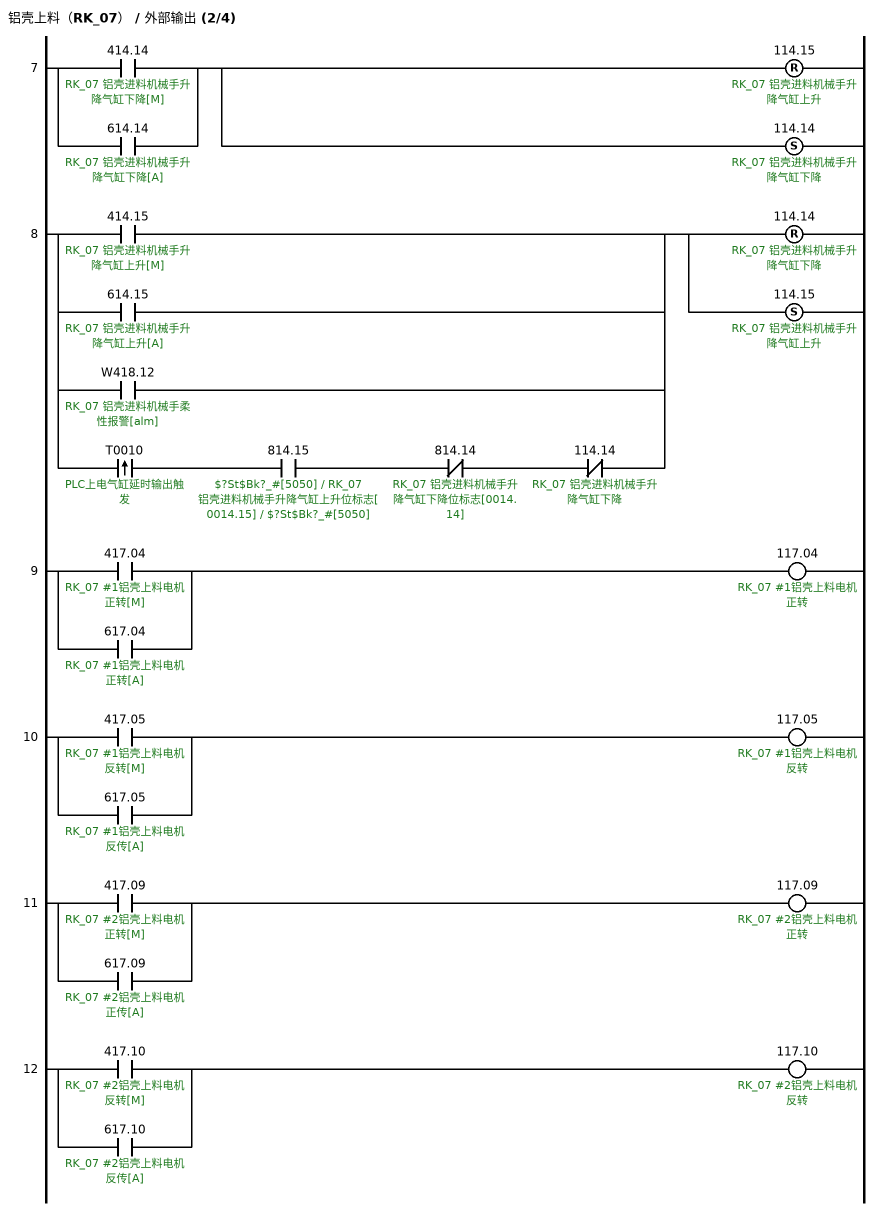
; rung 7
LD 414.14  ; RK_07 铝壳进料机械手升降气缸下降[M]
OR 614.14  ; RK_07 铝壳进料机械手升降气缸下降[A]
RSET 114.15  ; RK_07 铝壳进料机械手升降气缸上升
SET 114.14  ; RK_07 铝壳进料机械手升降气缸下降
; rung 8
LD 414.15  ; RK_07 铝壳进料机械手升降气缸上升[M]
OR 614.15  ; RK_07 铝壳进料机械手升降气缸上升[A]
OR W418.12  ; RK_07 铝壳进料机械手柔性报警[alm]
@LD T0010  ; PLC上电气缸延时输出触发
AND 814.15  ; $?St$Bk?_#[5050] / RK_07 铝壳进料机械手升降气缸上升位标志[0014.15] / $?St$Bk?_#[5050]
ANDNOT 814.14  ; RK_07 铝壳进料机械手升降气缸下降位标志[0014.14]
ANDNOT 114.14  ; RK_07 铝壳进料机械手升降气缸下降
ORLD
RSET 114.14  ; RK_07 铝壳进料机械手升降气缸下降
SET 114.15  ; RK_07 铝壳进料机械手升降气缸上升
; rung 9
LD 417.04  ; RK_07 #1铝壳上料电机正转[M]
OR 617.04  ; RK_07 #1铝壳上料电机正转[A]
OUT 117.04  ; RK_07 #1铝壳上料电机正转
; rung 10
LD 417.05  ; RK_07 #1铝壳上料电机反转[M]
OR 617.05  ; RK_07 #1铝壳上料电机反传[A]
OUT 117.05  ; RK_07 #1铝壳上料电机反转
; rung 11
LD 417.09  ; RK_07 #2铝壳上料电机正转[M]
OR 617.09  ; RK_07 #2铝壳上料电机正传[A]
OUT 117.09  ; RK_07 #2铝壳上料电机正转
; rung 12
LD 417.10  ; RK_07 #2铝壳上料电机反转[M]
OR 617.10  ; RK_07 #2铝壳上料电机反传[A]
OUT 117.10  ; RK_07 #2铝壳上料电机反转

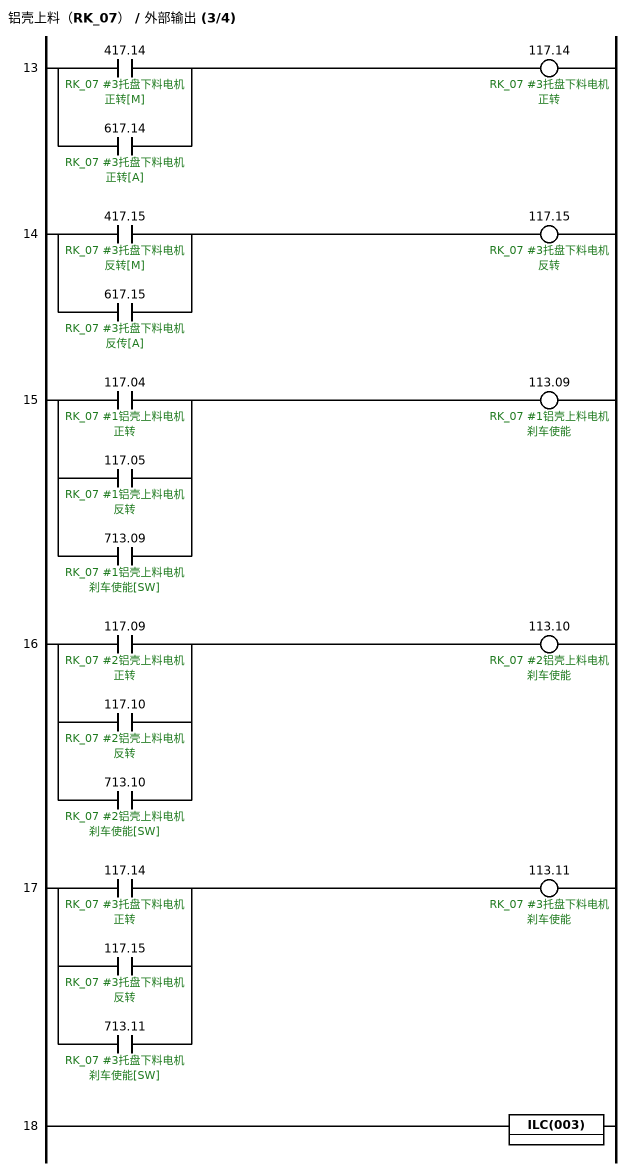
; rung 13
LD 417.14  ; RK_07 #3托盘下料电机正转[M]
OR 617.14  ; RK_07 #3托盘下料电机正转[A]
OUT 117.14  ; RK_07 #3托盘下料电机正转
; rung 14
LD 417.15  ; RK_07 #3托盘下料电机反转[M]
OR 617.15  ; RK_07 #3托盘下料电机反传[A]
OUT 117.15  ; RK_07 #3托盘下料电机反转
; rung 15
LD 117.04  ; RK_07 #1铝壳上料电机正转
OR 117.05  ; RK_07 #1铝壳上料电机反转
OR 713.09  ; RK_07 #1铝壳上料电机刹车使能[SW]
OUT 113.09  ; RK_07 #1铝壳上料电机刹车使能
; rung 16
LD 117.09  ; RK_07 #2铝壳上料电机正转
OR 117.10  ; RK_07 #2铝壳上料电机反转
OR 713.10  ; RK_07 #2铝壳上料电机刹车使能[SW]
OUT 113.10  ; RK_07 #2铝壳上料电机刹车使能
; rung 17
LD 117.14  ; RK_07 #3托盘下料电机正转
OR 117.15  ; RK_07 #3托盘下料电机反转
OR 713.11  ; RK_07 #3托盘下料电机刹车使能[SW]
OUT 113.11  ; RK_07 #3托盘下料电机刹车使能
; rung 18
ILC(003)

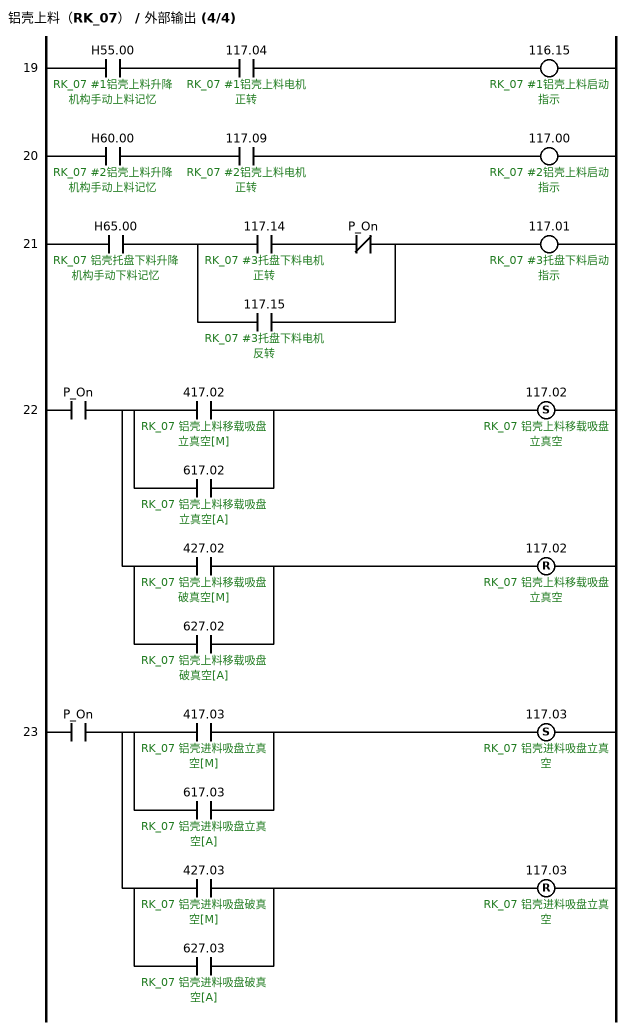
; rung 19
LD H55.00  ; RK_07 #1铝壳上料升降机构手动上料记忆
AND 117.04  ; RK_07 #1铝壳上料电机正转
OUT 116.15  ; RK_07 #1铝壳上料启动指示
; rung 20
LD H60.00  ; RK_07 #2铝壳上料升降机构手动上料记忆
AND 117.09  ; RK_07 #2铝壳上料电机正转
OUT 117.00  ; RK_07 #2铝壳上料启动指示
; rung 21
LD H65.00  ; RK_07 铝壳托盘下料升降机构手动下料记忆
LD 117.14  ; RK_07 #3托盘下料电机正转
ANDNOT P_On
OR 117.15  ; RK_07 #3托盘下料电机反转
ANDLD
OUT 117.01  ; RK_07 #3托盘下料启动指示
; rung 22
LD P_On
OUT TR0
LD 417.02  ; RK_07 铝壳上料移载吸盘立真空[M]
OR 617.02  ; RK_07 铝壳上料移载吸盘立真空[A]
ANDLD
SET 117.02  ; RK_07 铝壳上料移载吸盘立真空
LD TR0
LD 427.02  ; RK_07 铝壳上料移载吸盘破真空[M]
OR 627.02  ; RK_07 铝壳上料移载吸盘破真空[A]
ANDLD
RSET 117.02  ; RK_07 铝壳上料移载吸盘立真空
; rung 23
LD P_On
OUT TR0
LD 417.03  ; RK_07 铝壳进料吸盘立真空[M]
OR 617.03  ; RK_07 铝壳进料吸盘立真空[A]
ANDLD
SET 117.03  ; RK_07 铝壳进料吸盘立真空
LD TR0
LD 427.03  ; RK_07 铝壳进料吸盘破真空[M]
OR 627.03  ; RK_07 铝壳进料吸盘破真空[A]
ANDLD
RSET 117.03  ; RK_07 铝壳进料吸盘立真空

### Section END
; rung 0
END(001)

## Program 铝壳除尘_RK_08 (cyclic task 8)

### Section Main

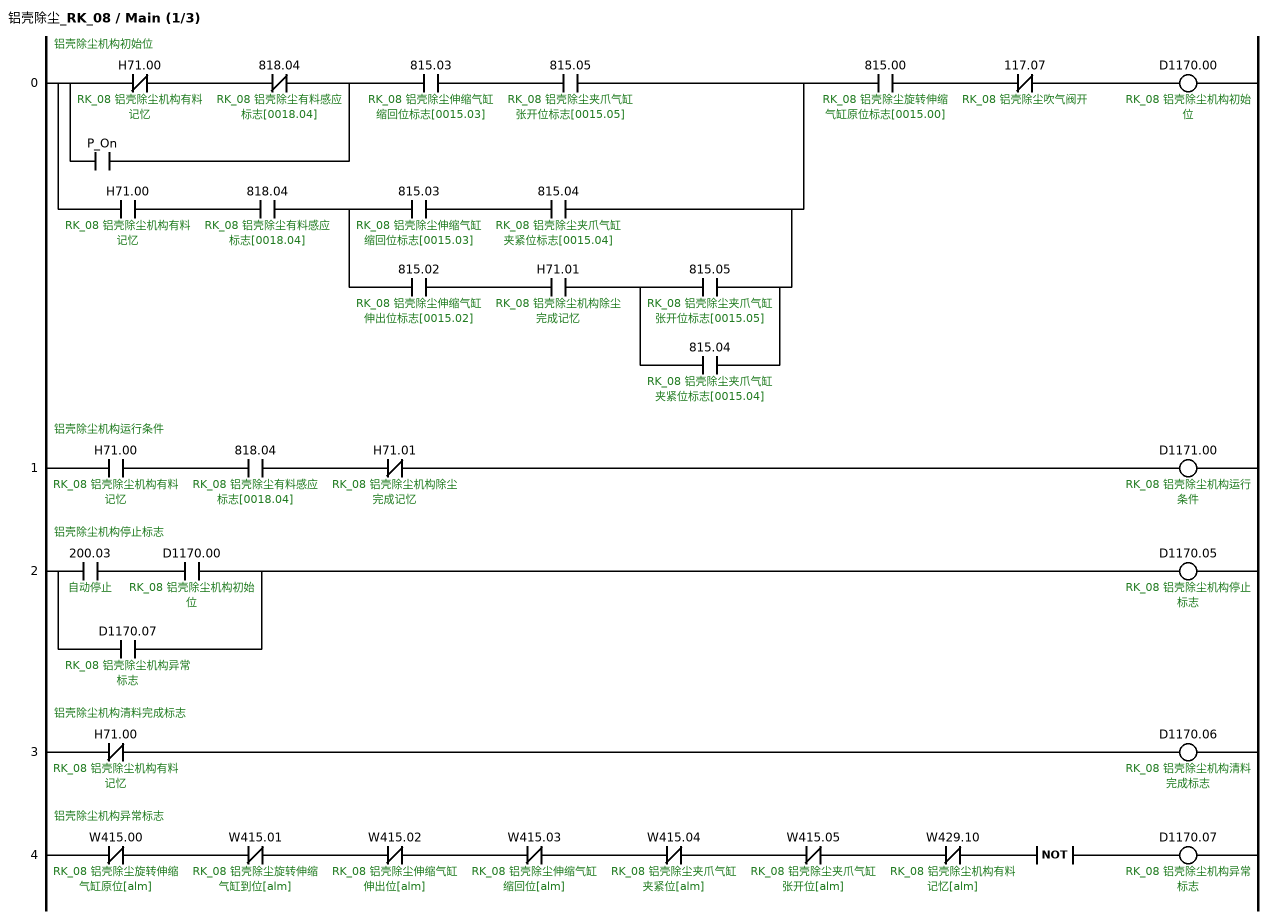
; rung 0: 铝壳除尘机构初始位
LDNOT H71.00  ; RK_08 铝壳除尘机构有料记忆
ANDNOT 818.04  ; RK_08 铝壳除尘有料感应标志[0018.04]
OR P_On
AND 815.03  ; RK_08 铝壳除尘伸缩气缸缩回位标志[0015.03]
AND 815.05  ; RK_08 铝壳除尘夹爪气缸张开位标志[0015.05]
LD H71.00  ; RK_08 铝壳除尘机构有料记忆
AND 818.04  ; RK_08 铝壳除尘有料感应标志[0018.04]
LD 815.03  ; RK_08 铝壳除尘伸缩气缸缩回位标志[0015.03]
AND 815.04  ; RK_08 铝壳除尘夹爪气缸夹紧位标志[0015.04]
LD 815.02  ; RK_08 铝壳除尘伸缩气缸伸出位标志[0015.02]
AND H71.01  ; RK_08 铝壳除尘机构除尘完成记忆
LD 815.05  ; RK_08 铝壳除尘夹爪气缸张开位标志[0015.05]
OR 815.04  ; RK_08 铝壳除尘夹爪气缸夹紧位标志[0015.04]
ANDLD
ORLD
ANDLD
ORLD
AND 815.00  ; RK_08 铝壳除尘旋转伸缩气缸原位标志[0015.00]
ANDNOT 117.07  ; RK_08 铝壳除尘吹气阀开
OUT D1170.00  ; RK_08 铝壳除尘机构初始位
; rung 1: 铝壳除尘机构运行条件
LD H71.00  ; RK_08 铝壳除尘机构有料记忆
AND 818.04  ; RK_08 铝壳除尘有料感应标志[0018.04]
ANDNOT H71.01  ; RK_08 铝壳除尘机构除尘完成记忆
OUT D1171.00  ; RK_08 铝壳除尘机构运行条件
; rung 2: 铝壳除尘机构停止标志
LD 200.03  ; 自动停止
AND D1170.00  ; RK_08 铝壳除尘机构初始位
OR D1170.07  ; RK_08 铝壳除尘机构异常标志
OUT D1170.05  ; RK_08 铝壳除尘机构停止标志
; rung 3: 铝壳除尘机构清料完成标志
LDNOT H71.00  ; RK_08 铝壳除尘机构有料记忆
OUT D1170.06  ; RK_08 铝壳除尘机构清料完成标志
; rung 4: 铝壳除尘机构异常标志
LDNOT W415.00  ; RK_08 铝壳除尘旋转伸缩气缸原位[alm]
ANDNOT W415.01  ; RK_08 铝壳除尘旋转伸缩气缸到位[alm]
ANDNOT W415.02  ; RK_08 铝壳除尘伸缩气缸伸出位[alm]
ANDNOT W415.03  ; RK_08 铝壳除尘伸缩气缸缩回位[alm]
ANDNOT W415.04  ; RK_08 铝壳除尘夹爪气缸夹紧位[alm]
ANDNOT W415.05  ; RK_08 铝壳除尘夹爪气缸张开位[alm]
ANDNOT W429.10  ; RK_08 铝壳除尘机构有料记忆[alm]
NOT(520)
OUT D1170.07  ; RK_08 铝壳除尘机构异常标志

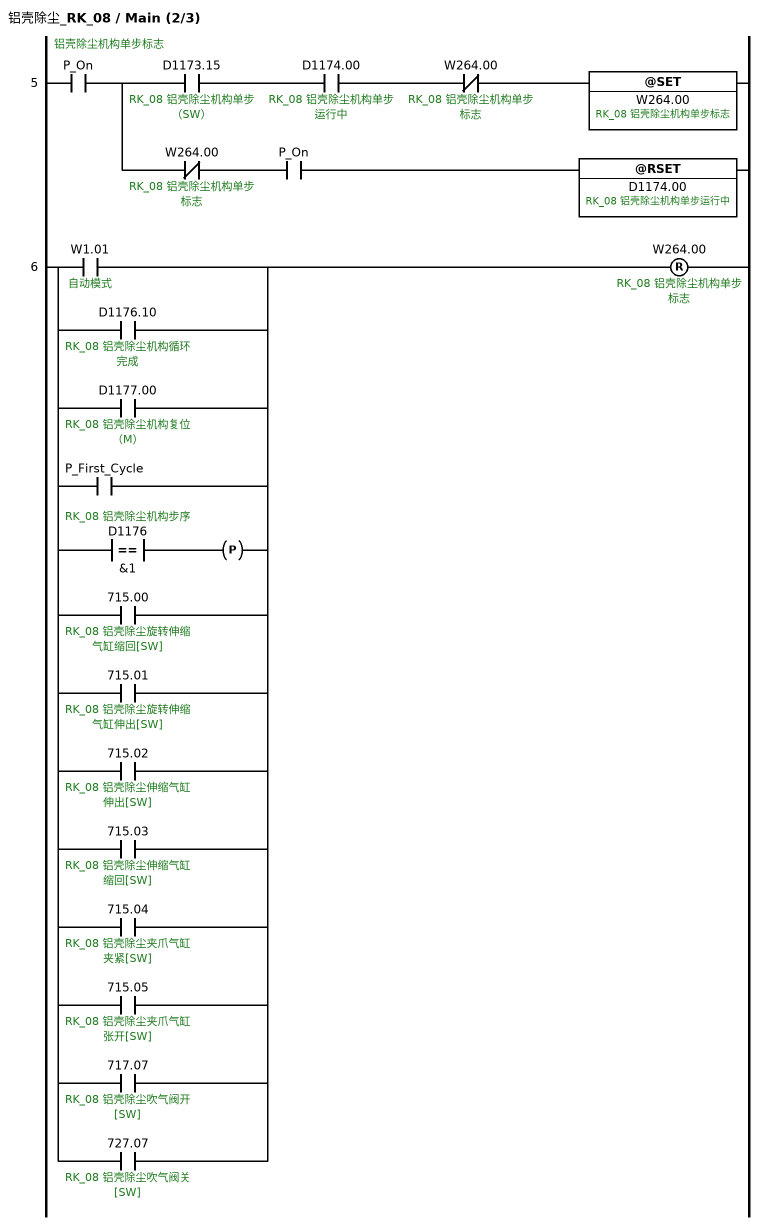
; rung 5: 铝壳除尘机构单步标志
LD P_On
OUT TR0
AND D1173.15  ; RK_08 铝壳除尘机构单步（SW）
AND D1174.00  ; RK_08 铝壳除尘机构单步运行中
ANDNOT W264.00  ; RK_08 铝壳除尘机构单步标志
@SET W264.00  ; RK_08 铝壳除尘机构单步标志
LD TR0
ANDNOT W264.00  ; RK_08 铝壳除尘机构单步标志
AND P_On
@RSET D1174.00  ; RK_08 铝壳除尘机构单步运行中
; rung 6
LD W1.01  ; 自动模式
OR D1176.10  ; RK_08 铝壳除尘机构循环完成
OR D1177.00  ; RK_08 铝壳除尘机构复位（M）
OR P_First_Cycle
LD=(300) D1176 &1  ; RK_08 铝壳除尘机构步序
UP(521)
ORLD
LD 715.00  ; RK_08 铝壳除尘旋转伸缩气缸缩回[SW]
OR 715.01  ; RK_08 铝壳除尘旋转伸缩气缸伸出[SW]
OR 715.02  ; RK_08 铝壳除尘伸缩气缸伸出[SW]
OR 715.03  ; RK_08 铝壳除尘伸缩气缸缩回[SW]
OR 715.04  ; RK_08 铝壳除尘夹爪气缸夹紧[SW]
OR 715.05  ; RK_08 铝壳除尘夹爪气缸张开[SW]
OR 717.07  ; RK_08 铝壳除尘吹气阀开[SW]
OR 727.07  ; RK_08 铝壳除尘吹气阀关[SW]
ORLD
RSET W264.00  ; RK_08 铝壳除尘机构单步标志

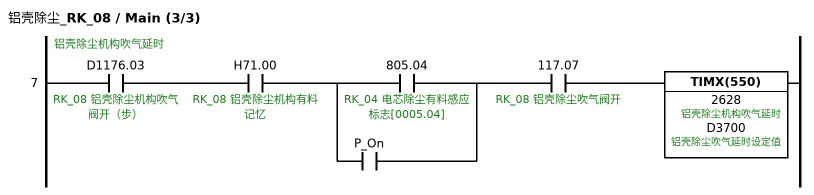
; rung 7: 铝壳除尘机构吹气延时
LD D1176.03  ; RK_08 铝壳除尘机构吹气阀开（步）
AND H71.00  ; RK_08 铝壳除尘机构有料记忆
LD 805.04  ; RK_04 电芯除尘有料感应标志[0005.04]
OR P_On
ANDLD
AND 117.07  ; RK_08 铝壳除尘吹气阀开
TIMX(550) 2628 D3700  ; 铝壳除尘吹气延时设定值, 铝壳除尘机构吹气延时

### Section 手动

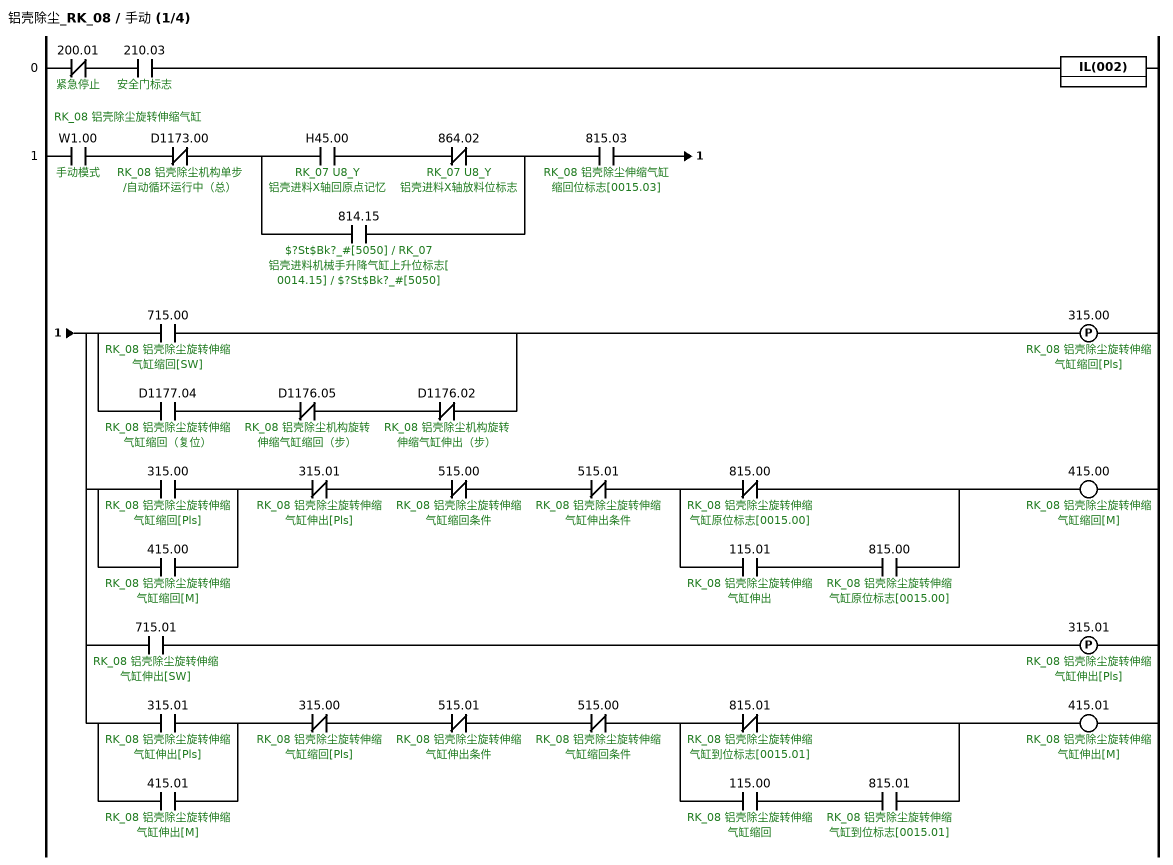
; rung 0
LDNOT 200.01  ; 紧急停止
AND 210.03  ; 安全门标志
IL(002)
; rung 1: RK_08 铝壳除尘旋转伸缩气缸
LD W1.00  ; 手动模式
ANDNOT D1173.00  ; RK_08 铝壳除尘机构单步/自动循环运行中（总）
LD H45.00  ; RK_07 U8_Y 铝壳进料X轴回原点记忆
ANDNOT 864.02  ; RK_07 U8_Y 铝壳进料X轴放料位标志
OR 814.15  ; $?St$Bk?_#[5050] / RK_07 铝壳进料机械手升降气缸上升位标志[0014.15] / $?St$Bk?_#[5050]
ANDLD
AND 815.03  ; RK_08 铝壳除尘伸缩气缸缩回位标志[0015.03]
OUT TR0
LD 715.00  ; RK_08 铝壳除尘旋转伸缩气缸缩回[SW]
LD D1177.04  ; RK_08 铝壳除尘旋转伸缩气缸缩回（复位）
ANDNOT D1176.05  ; RK_08 铝壳除尘机构旋转伸缩气缸缩回（步）
ANDNOT D1176.02  ; RK_08 铝壳除尘机构旋转伸缩气缸伸出（步）
ORLD
ANDLD
DIFU(013) 315.00  ; RK_08 铝壳除尘旋转伸缩气缸缩回[Pls]
LD TR0
LD 315.00  ; RK_08 铝壳除尘旋转伸缩气缸缩回[Pls]
OR 415.00  ; RK_08 铝壳除尘旋转伸缩气缸缩回[M]
ANDLD
ANDNOT 315.01  ; RK_08 铝壳除尘旋转伸缩气缸伸出[Pls]
ANDNOT 515.00  ; RK_08 铝壳除尘旋转伸缩气缸缩回条件
ANDNOT 515.01  ; RK_08 铝壳除尘旋转伸缩气缸伸出条件
LDNOT 815.00  ; RK_08 铝壳除尘旋转伸缩气缸原位标志[0015.00]
LD 115.01  ; RK_08 铝壳除尘旋转伸缩气缸伸出
AND 815.00  ; RK_08 铝壳除尘旋转伸缩气缸原位标志[0015.00]
ORLD
ANDLD
OUT 415.00  ; RK_08 铝壳除尘旋转伸缩气缸缩回[M]
LD TR0
AND 715.01  ; RK_08 铝壳除尘旋转伸缩气缸伸出[SW]
DIFU(013) 315.01  ; RK_08 铝壳除尘旋转伸缩气缸伸出[Pls]
LD TR0
LD 315.01  ; RK_08 铝壳除尘旋转伸缩气缸伸出[Pls]
OR 415.01  ; RK_08 铝壳除尘旋转伸缩气缸伸出[M]
ANDLD
ANDNOT 315.00  ; RK_08 铝壳除尘旋转伸缩气缸缩回[Pls]
ANDNOT 515.01  ; RK_08 铝壳除尘旋转伸缩气缸伸出条件
ANDNOT 515.00  ; RK_08 铝壳除尘旋转伸缩气缸缩回条件
LDNOT 815.01  ; RK_08 铝壳除尘旋转伸缩气缸到位标志[0015.01]
LD 115.00  ; RK_08 铝壳除尘旋转伸缩气缸缩回
AND 815.01  ; RK_08 铝壳除尘旋转伸缩气缸到位标志[0015.01]
ORLD
ANDLD
OUT 415.01  ; RK_08 铝壳除尘旋转伸缩气缸伸出[M]

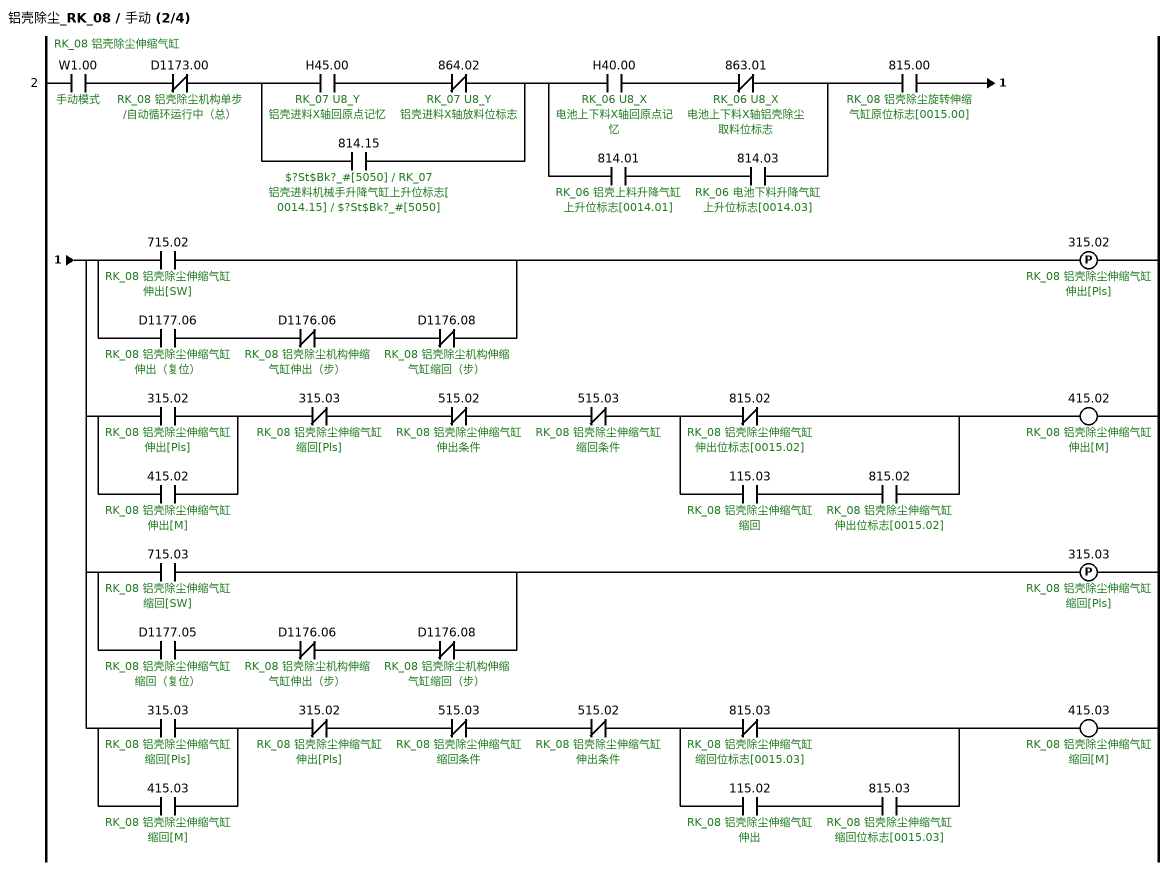
; rung 2: RK_08 铝壳除尘伸缩气缸
LD W1.00  ; 手动模式
ANDNOT D1173.00  ; RK_08 铝壳除尘机构单步/自动循环运行中（总）
LD H45.00  ; RK_07 U8_Y 铝壳进料X轴回原点记忆
ANDNOT 864.02  ; RK_07 U8_Y 铝壳进料X轴放料位标志
OR 814.15  ; $?St$Bk?_#[5050] / RK_07 铝壳进料机械手升降气缸上升位标志[0014.15] / $?St$Bk?_#[5050]
ANDLD
LD H40.00  ; RK_06 U8_X 电池上下料X轴回原点记忆
ANDNOT 863.01  ; RK_06 U8_X 电池上下料X轴铝壳除尘取料位标志
LD 814.01  ; RK_06 铝壳上料升降气缸上升位标志[0014.01]
AND 814.03  ; RK_06 电池下料升降气缸上升位标志[0014.03]
ORLD
ANDLD
AND 815.00  ; RK_08 铝壳除尘旋转伸缩气缸原位标志[0015.00]
OUT TR0
LD 715.02  ; RK_08 铝壳除尘伸缩气缸伸出[SW]
LD D1177.06  ; RK_08 铝壳除尘伸缩气缸伸出（复位）
ANDNOT D1176.06  ; RK_08 铝壳除尘机构伸缩气缸伸出（步）
ANDNOT D1176.08  ; RK_08 铝壳除尘机构伸缩气缸缩回（步）
ORLD
ANDLD
DIFU(013) 315.02  ; RK_08 铝壳除尘伸缩气缸伸出[Pls]
LD TR0
LD 315.02  ; RK_08 铝壳除尘伸缩气缸伸出[Pls]
OR 415.02  ; RK_08 铝壳除尘伸缩气缸伸出[M]
ANDLD
ANDNOT 315.03  ; RK_08 铝壳除尘伸缩气缸缩回[Pls]
ANDNOT 515.02  ; RK_08 铝壳除尘伸缩气缸伸出条件
ANDNOT 515.03  ; RK_08 铝壳除尘伸缩气缸缩回条件
LDNOT 815.02  ; RK_08 铝壳除尘伸缩气缸伸出位标志[0015.02]
LD 115.03  ; RK_08 铝壳除尘伸缩气缸缩回
AND 815.02  ; RK_08 铝壳除尘伸缩气缸伸出位标志[0015.02]
ORLD
ANDLD
OUT 415.02  ; RK_08 铝壳除尘伸缩气缸伸出[M]
LD TR0
LD 715.03  ; RK_08 铝壳除尘伸缩气缸缩回[SW]
LD D1177.05  ; RK_08 铝壳除尘伸缩气缸缩回（复位）
ANDNOT D1176.06  ; RK_08 铝壳除尘机构伸缩气缸伸出（步）
ANDNOT D1176.08  ; RK_08 铝壳除尘机构伸缩气缸缩回（步）
ORLD
ANDLD
DIFU(013) 315.03  ; RK_08 铝壳除尘伸缩气缸缩回[Pls]
LD TR0
LD 315.03  ; RK_08 铝壳除尘伸缩气缸缩回[Pls]
OR 415.03  ; RK_08 铝壳除尘伸缩气缸缩回[M]
ANDLD
ANDNOT 315.02  ; RK_08 铝壳除尘伸缩气缸伸出[Pls]
ANDNOT 515.03  ; RK_08 铝壳除尘伸缩气缸缩回条件
ANDNOT 515.02  ; RK_08 铝壳除尘伸缩气缸伸出条件
LDNOT 815.03  ; RK_08 铝壳除尘伸缩气缸缩回位标志[0015.03]
LD 115.02  ; RK_08 铝壳除尘伸缩气缸伸出
AND 815.03  ; RK_08 铝壳除尘伸缩气缸缩回位标志[0015.03]
ORLD
ANDLD
OUT 415.03  ; RK_08 铝壳除尘伸缩气缸缩回[M]

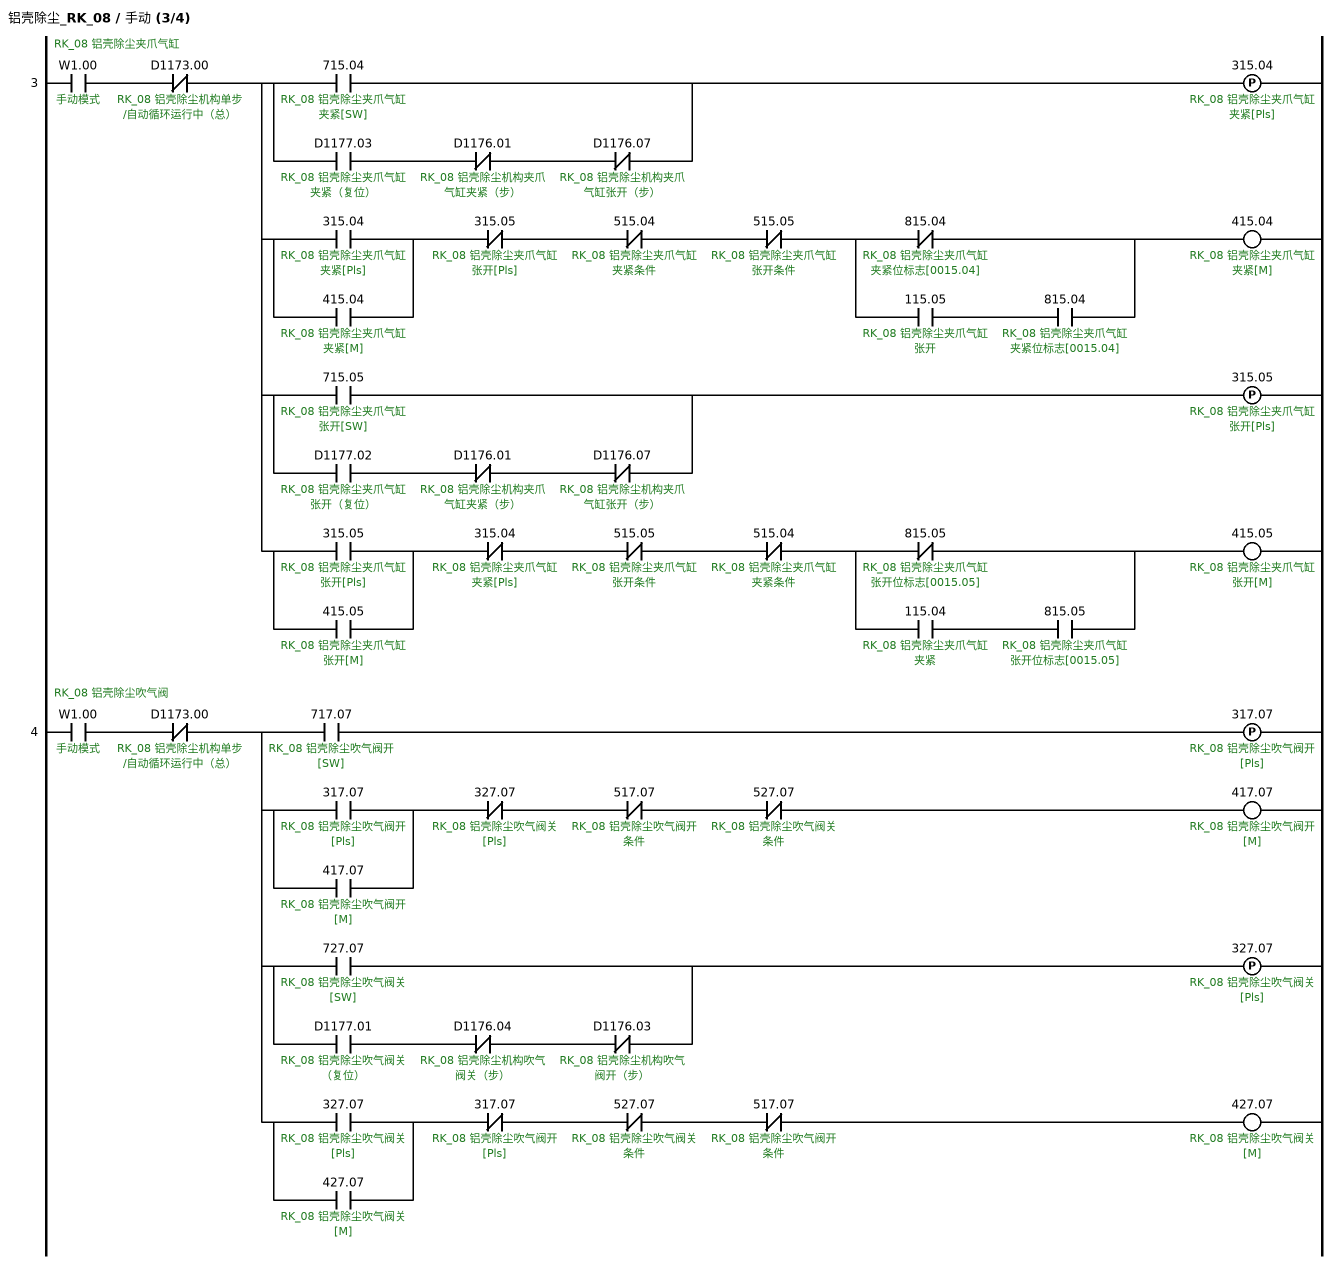
; rung 3: RK_08 铝壳除尘夹爪气缸
LD W1.00  ; 手动模式
ANDNOT D1173.00  ; RK_08 铝壳除尘机构单步/自动循环运行中（总）
OUT TR0
LD 715.04  ; RK_08 铝壳除尘夹爪气缸夹紧[SW]
LD D1177.03  ; RK_08 铝壳除尘夹爪气缸夹紧（复位）
ANDNOT D1176.01  ; RK_08 铝壳除尘机构夹爪气缸夹紧（步）
ANDNOT D1176.07  ; RK_08 铝壳除尘机构夹爪气缸张开（步）
ORLD
ANDLD
DIFU(013) 315.04  ; RK_08 铝壳除尘夹爪气缸夹紧[Pls]
LD TR0
LD 315.04  ; RK_08 铝壳除尘夹爪气缸夹紧[Pls]
OR 415.04  ; RK_08 铝壳除尘夹爪气缸夹紧[M]
ANDLD
ANDNOT 315.05  ; RK_08 铝壳除尘夹爪气缸张开[Pls]
ANDNOT 515.04  ; RK_08 铝壳除尘夹爪气缸夹紧条件
ANDNOT 515.05  ; RK_08 铝壳除尘夹爪气缸张开条件
LDNOT 815.04  ; RK_08 铝壳除尘夹爪气缸夹紧位标志[0015.04]
LD 115.05  ; RK_08 铝壳除尘夹爪气缸张开
AND 815.04  ; RK_08 铝壳除尘夹爪气缸夹紧位标志[0015.04]
ORLD
ANDLD
OUT 415.04  ; RK_08 铝壳除尘夹爪气缸夹紧[M]
LD TR0
LD 715.05  ; RK_08 铝壳除尘夹爪气缸张开[SW]
LD D1177.02  ; RK_08 铝壳除尘夹爪气缸张开（复位）
ANDNOT D1176.01  ; RK_08 铝壳除尘机构夹爪气缸夹紧（步）
ANDNOT D1176.07  ; RK_08 铝壳除尘机构夹爪气缸张开（步）
ORLD
ANDLD
DIFU(013) 315.05  ; RK_08 铝壳除尘夹爪气缸张开[Pls]
LD TR0
LD 315.05  ; RK_08 铝壳除尘夹爪气缸张开[Pls]
OR 415.05  ; RK_08 铝壳除尘夹爪气缸张开[M]
ANDLD
ANDNOT 315.04  ; RK_08 铝壳除尘夹爪气缸夹紧[Pls]
ANDNOT 515.05  ; RK_08 铝壳除尘夹爪气缸张开条件
ANDNOT 515.04  ; RK_08 铝壳除尘夹爪气缸夹紧条件
LDNOT 815.05  ; RK_08 铝壳除尘夹爪气缸张开位标志[0015.05]
LD 115.04  ; RK_08 铝壳除尘夹爪气缸夹紧
AND 815.05  ; RK_08 铝壳除尘夹爪气缸张开位标志[0015.05]
ORLD
ANDLD
OUT 415.05  ; RK_08 铝壳除尘夹爪气缸张开[M]
; rung 4: RK_08 铝壳除尘吹气阀
LD W1.00  ; 手动模式
ANDNOT D1173.00  ; RK_08 铝壳除尘机构单步/自动循环运行中（总）
OUT TR0
AND 717.07  ; RK_08 铝壳除尘吹气阀开[SW]
DIFU(013) 317.07  ; RK_08 铝壳除尘吹气阀开[Pls]
LD TR0
LD 317.07  ; RK_08 铝壳除尘吹气阀开[Pls]
OR 417.07  ; RK_08 铝壳除尘吹气阀开[M]
ANDLD
ANDNOT 327.07  ; RK_08 铝壳除尘吹气阀关[Pls]
ANDNOT 517.07  ; RK_08 铝壳除尘吹气阀开条件
ANDNOT 527.07  ; RK_08 铝壳除尘吹气阀关条件
OUT 417.07  ; RK_08 铝壳除尘吹气阀开[M]
LD TR0
LD 727.07  ; RK_08 铝壳除尘吹气阀关[SW]
LD D1177.01  ; RK_08 铝壳除尘吹气阀关（复位）
ANDNOT D1176.04  ; RK_08 铝壳除尘机构吹气阀关（步）
ANDNOT D1176.03  ; RK_08 铝壳除尘机构吹气阀开（步）
ORLD
ANDLD
DIFU(013) 327.07  ; RK_08 铝壳除尘吹气阀关[Pls]
LD TR0
LD 327.07  ; RK_08 铝壳除尘吹气阀关[Pls]
OR 427.07  ; RK_08 铝壳除尘吹气阀关[M]
ANDLD
ANDNOT 317.07  ; RK_08 铝壳除尘吹气阀开[Pls]
ANDNOT 527.07  ; RK_08 铝壳除尘吹气阀关条件
ANDNOT 517.07  ; RK_08 铝壳除尘吹气阀开条件
OUT 427.07  ; RK_08 铝壳除尘吹气阀关[M]

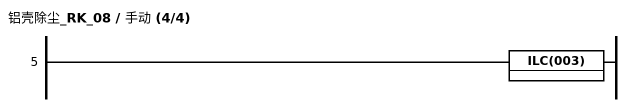
; rung 5
ILC(003)

### Section 自动

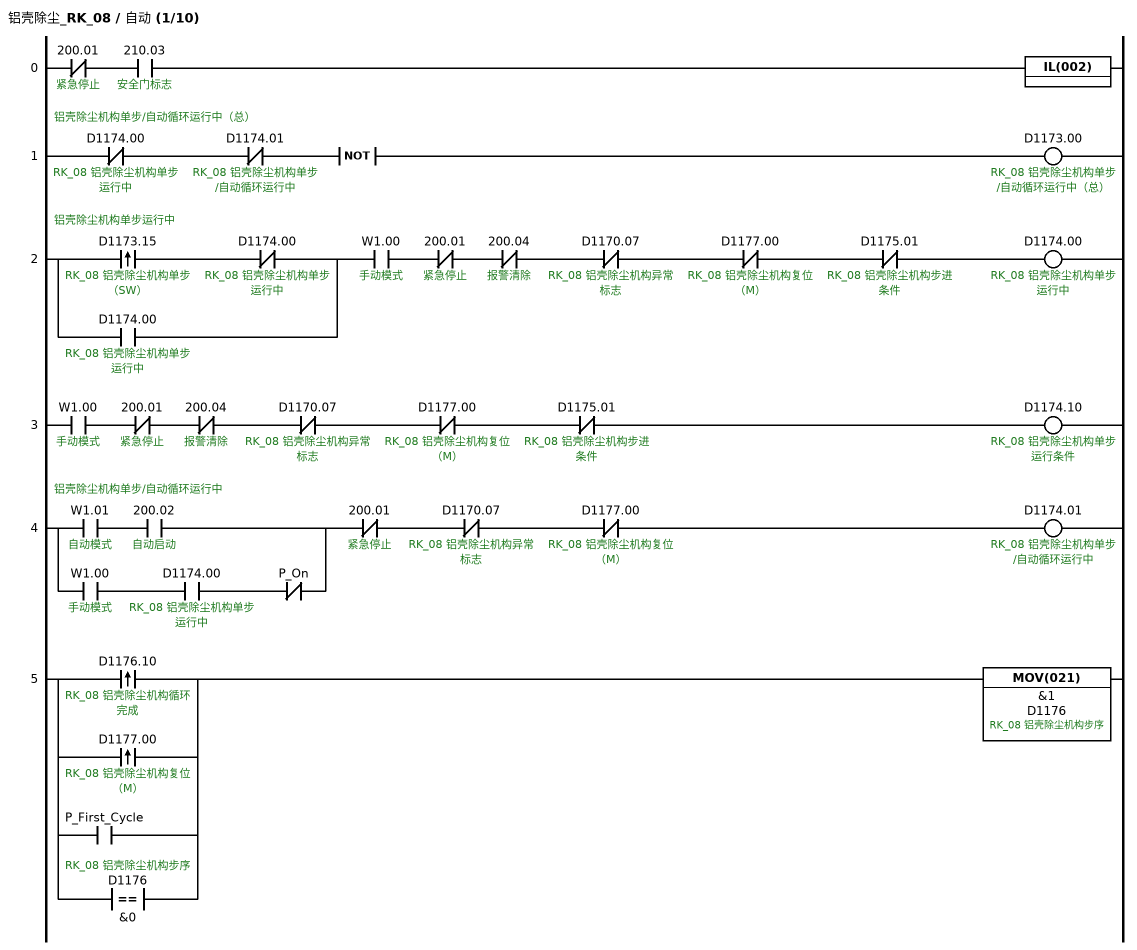
; rung 0
LDNOT 200.01  ; 紧急停止
AND 210.03  ; 安全门标志
IL(002)
; rung 1: 铝壳除尘机构单步/自动循环运行中（总）
LDNOT D1174.00  ; RK_08 铝壳除尘机构单步运行中
ANDNOT D1174.01  ; RK_08 铝壳除尘机构单步/自动循环运行中
NOT(520)
OUT D1173.00  ; RK_08 铝壳除尘机构单步/自动循环运行中（总）
; rung 2: 铝壳除尘机构单步运行中
@LD D1173.15  ; RK_08 铝壳除尘机构单步（SW）
ANDNOT D1174.00  ; RK_08 铝壳除尘机构单步运行中
OR D1174.00  ; RK_08 铝壳除尘机构单步运行中
AND W1.00  ; 手动模式
ANDNOT 200.01  ; 紧急停止
ANDNOT 200.04  ; 报警清除
ANDNOT D1170.07  ; RK_08 铝壳除尘机构异常标志
ANDNOT D1177.00  ; RK_08 铝壳除尘机构复位（M）
ANDNOT D1175.01  ; RK_08 铝壳除尘机构步进条件
OUT D1174.00  ; RK_08 铝壳除尘机构单步运行中
; rung 3
LD W1.00  ; 手动模式
ANDNOT 200.01  ; 紧急停止
ANDNOT 200.04  ; 报警清除
ANDNOT D1170.07  ; RK_08 铝壳除尘机构异常标志
ANDNOT D1177.00  ; RK_08 铝壳除尘机构复位（M）
ANDNOT D1175.01  ; RK_08 铝壳除尘机构步进条件
OUT D1174.10  ; RK_08 铝壳除尘机构单步运行条件
; rung 4: 铝壳除尘机构单步/自动循环运行中
LD W1.01  ; 自动模式
AND 200.02  ; 自动启动
LD W1.00  ; 手动模式
AND D1174.00  ; RK_08 铝壳除尘机构单步运行中
ANDNOT P_On
ORLD
ANDNOT 200.01  ; 紧急停止
ANDNOT D1170.07  ; RK_08 铝壳除尘机构异常标志
ANDNOT D1177.00  ; RK_08 铝壳除尘机构复位（M）
OUT D1174.01  ; RK_08 铝壳除尘机构单步/自动循环运行中
; rung 5
@LD D1176.10  ; RK_08 铝壳除尘机构循环完成
@OR D1177.00  ; RK_08 铝壳除尘机构复位（M）
OR P_First_Cycle
OR=(300) D1176 &0  ; RK_08 铝壳除尘机构步序
MOV(021) &1 D1176  ; RK_08 铝壳除尘机构步序

